SPLINE
SPL {X  -103.775, Y  +255.731, Z    +0.000, E1   +56.205, E3 +52331.695}
SPL {X  -141.196, Y  +302.265, Z    +0.000, E1   +49.914, E3 +52369.180}
SPL {X  -155.405, Y  +339.473, Z    +0.000, E1   +34.418, E3 +52378.880}
SPL {X  -159.172, Y  +361.346, Z    +0.000, E1   +18.323, E3 +52381.305}
SPL {X  -159.962, Y  +374.520, Z    +0.000, E1    +5.534, E3 +52381.918}
SPL {X  -159.990, Y  +379.490, Z    +0.000, E1    +0.023, E3 +52381.975}
SPL {X  -159.990, Y  +381.667, Z    +0.000, E1    -4.707, E3 +52381.997}
SPL {X  -159.990, Y  +385.814, Z    +0.000, E1   -15.621, E3 +52382.101}
SPL {X  -159.990, Y  +390.948, Z    +0.000, E1   -28.850, E3 +52382.377}
SPL {X  -159.990, Y  +399.006, Z    +0.000, E1   -45.565, E3 +52383.089}
SPL {X  -159.990, Y  +410.008, Z    +0.000, E1   -58.546, E3 +52384.699}
SPL {X  -159.990, Y  +426.664, Z    +0.000, E1   -66.963, E3 +52388.320}
SPL {X  -159.990, Y  +494.829, Z    +0.000, E1   -73.764, E3 +52410.084}
SPL {X  -158.798, Y  +695.991, Z    +0.000, E1   -74.986, E3 +52500.017}
SPL {X  -156.512, Y  +709.677, Z    +0.000, E1   -74.772, E3 +52510.161}
SPL {X  -153.684, Y  +720.975, Z    +0.000, E1   -74.508, E3 +52519.448}
SPL {X  -149.353, Y  +733.863, Z    +0.000, E1   -74.100, E3 +52531.036}
SPL {X  -145.190, Y  +743.705, Z    +0.000, E1   -73.640, E3 +52540.717}
SPL {X  -141.940, Y  +750.322, Z    +0.000, E1   -73.290, E3 +52547.484}
SPL {X  -138.555, Y  +756.496, Z    +0.000, E1   -72.905, E3 +52554.049}
SPL {X  -135.025, Y  +762.319, Z    +0.000, E1   -72.483, E3 +52560.428}
SPL {X  -131.747, Y  +767.272, Z    +0.000, E1   -72.071, E3 +52565.953}
SPL {X  -128.648, Y  +771.613, Z    +0.000, E1   -71.666, E3 +52570.845}
SPL {X  -125.012, Y  +776.344, Z    +0.000, E1   -71.184, E3 +52576.157}
SPL {X  -121.578, Y  +780.498, Z    +0.000, E1   -70.681, E3 +52580.800}
SPL {X  -119.460, Y  +782.925, Z    +0.000, E1   -70.353, E3 +52583.464}
SPL {X   -74.295, Y  +818.193, Z    +0.000, E1   -57.793, E3 +52692.125}
ENDSPLINE

SPLINE
SPL {X  -120.240, Y  +782.043, Z    +0.000, E1   -55.019, E3 +52890.621}
SPL {X  -145.777, Y  +742.423, Z    +0.000, E1   -46.722, E3 +52912.501}
SPL {X  -154.920, Y  +716.458, Z    +0.000, E1   -35.175, E3 +52918.556}
SPL {X  -159.063, Y  +693.702, Z    +0.000, E1   -19.028, E3 +52921.337}
SPL {X  -159.958, Y  +679.684, Z    +0.000, E1    -5.688, E3 +52922.049}
SPL {X  -159.990, Y  +674.512, Z    +0.000, E1    -0.026, E3 +52922.114}
SPL {X  -159.990, Y  +672.767, Z    +0.000, E1    +3.705, E3 +52922.127}
SPL {X  -159.990, Y  +669.310, Z    +0.000, E1   +12.444, E3 +52922.201}
SPL {X  -159.990, Y  +665.511, Z    +0.000, E1   +22.359, E3 +52922.360}
SPL {X  -159.990, Y  +658.432, Z    +0.000, E1   +38.720, E3 +52922.884}
SPL {X  -159.990, Y  +646.280, Z    +0.000, E1   +56.156, E3 +52924.413}
SPL {X  -159.990, Y  +625.549, Z    +0.000, E1   +67.208, E3 +52928.935}
SPL {X  -159.990, Y  +550.186, Z    +0.000, E1   +73.637, E3 +52954.340}
SPL {X  -159.493, Y  +364.902, Z    +0.000, E1   +74.541, E3 +53041.334}
SPL {X  -156.915, Y  +346.281, Z    +0.000, E1   +74.304, E3 +53054.930}
ENDSPLINE

SPLINE
SPL {X  -159.697, Y  +367.814, Z    +0.000, E1   +71.217, E3 +53072.248}
ENDSPLINE

SPLINE
SPL {X  -156.028, Y  +342.114, Z    +0.000, E1   +72.020, E3 +53082.402}
SPL {X  -150.925, Y  +324.412, Z    +0.000, E1   +72.419, E3 +53090.195}
SPL {X  -144.972, Y  +309.824, Z    +0.000, E1   +72.799, E3 +53095.797}
SPL {X  -139.605, Y  +299.351, Z    +0.000, E1   +73.035, E3 +53099.928}
SPL {X  -136.475, Y  +294.006, Z    +0.000, E1   +72.670, E3 +53105.713}
SPL {X  -133.214, Y  +288.895, Z    +0.000, E1   +72.272, E3 +53111.361}
SPL {X  -129.829, Y  +284.006, Z    +0.000, E1   +71.844, E3 +53116.836}
SPL {X  -126.314, Y  +279.309, Z    +0.000, E1   +71.374, E3 +53122.128}
SPL {X  -122.705, Y  +274.834, Z    +0.000, E1   +70.869, E3 +53127.139}
SPL {X  -119.804, Y  +271.463, Z    +0.000, E1   +70.429, E3 +53130.858}
SPL {X   -77.409, Y  +237.483, Z    +0.000, E1   +59.013, E3 +53224.534}
ENDSPLINE

SPLINE
SPL {X  -103.775, Y  +255.731, Z    +0.000, E1   +56.205, E3 +53421.247}
SPL {X  -133.021, Y  +288.605, Z    +0.000, E1   +53.007, E3 +53452.703}
SPL {X  -149.384, Y  +320.219, Z    +0.000, E1   +43.953, E3 +53464.427}
SPL {X  -157.534, Y  +349.577, Z    +0.000, E1   +27.748, E3 +53469.779}
SPL {X  -159.460, Y  +364.489, Z    +0.000, E1   +15.407, E3 +53471.074}
SPL {X  -159.962, Y  +374.520, Z    +0.000, E1    +5.534, E3 +53471.470}
SPL {X  -159.990, Y  +379.490, Z    +0.000, E1    +0.023, E3 +53471.527}
SPL {X  -159.990, Y  +381.667, Z    +0.000, E1    -4.707, E3 +53471.549}
SPL {X  -159.990, Y  +387.434, Z    +0.000, E1   -19.600, E3 +53471.732}
SPL {X  -159.990, Y  +392.971, Z    +0.000, E1   -33.903, E3 +53472.065}
SPL {X  -159.990, Y  +399.006, Z    +0.000, E1   -45.565, E3 +53472.641}
SPL {X  -159.990, Y  +410.008, Z    +0.000, E1   -58.546, E3 +53474.251}
SPL {X  -159.990, Y  +426.664, Z    +0.000, E1   -66.963, E3 +53477.872}
SPL {X  -159.990, Y  +494.829, Z    +0.000, E1   -73.764, E3 +53499.637}
SPL {X  -158.798, Y  +695.991, Z    +0.000, E1   -74.986, E3 +53589.569}
SPL {X  -156.512, Y  +709.677, Z    +0.000, E1   -74.772, E3 +53599.713}
SPL {X  -153.684, Y  +720.975, Z    +0.000, E1   -74.508, E3 +53609.000}
SPL {X  -149.353, Y  +733.863, Z    +0.000, E1   -74.100, E3 +53620.588}
SPL {X  -145.190, Y  +743.705, Z    +0.000, E1   -73.640, E3 +53630.269}
SPL {X  -141.940, Y  +750.322, Z    +0.000, E1   -73.290, E3 +53637.036}
SPL {X  -138.555, Y  +756.496, Z    +0.000, E1   -72.905, E3 +53643.601}
SPL {X  -135.025, Y  +762.319, Z    +0.000, E1   -72.483, E3 +53649.980}
SPL {X  -131.747, Y  +767.272, Z    +0.000, E1   -72.071, E3 +53655.505}
SPL {X  -127.432, Y  +773.236, Z    +0.000, E1   -71.530, E3 +53662.191}
SPL {X  -124.036, Y  +777.554, Z    +0.000, E1   -71.026, E3 +53667.089}
SPL {X  -120.782, Y  +781.422, Z    +0.000, E1   -70.584, E3 +53671.347}
SPL {X   -74.295, Y  +818.193, Z    +0.000, E1   -57.793, E3 +53781.678}
ENDSPLINE

SPLINE
SPL {X  -105.102, Y  +797.125, Z    +0.000, E1   -55.734, E3 +53961.044}
SPL {X  -126.361, Y  +774.631, Z    +0.000, E1   -54.192, E3 +53986.712}
SPL {X  -145.777, Y  +742.423, Z    +0.000, E1   -46.722, E3 +54002.053}
SPL {X  -154.920, Y  +716.458, Z    +0.000, E1   -35.175, E3 +54008.108}
SPL {X  -159.063, Y  +693.702, Z    +0.000, E1   -19.028, E3 +54010.889}
SPL {X  -159.958, Y  +679.684, Z    +0.000, E1    -5.688, E3 +54011.601}
SPL {X  -159.990, Y  +674.512, Z    +0.000, E1    -0.026, E3 +54011.666}
SPL {X  -159.990, Y  +672.767, Z    +0.000, E1    +3.705, E3 +54011.679}
SPL {X  -159.990, Y  +669.310, Z    +0.000, E1   +12.444, E3 +54011.753}
SPL {X  -159.990, Y  +665.511, Z    +0.000, E1   +22.359, E3 +54011.912}
SPL {X  -159.990, Y  +660.776, Z    +0.000, E1   +34.018, E3 +54012.218}
SPL {X  -159.990, Y  +655.863, Z    +0.000, E1   +43.768, E3 +54012.676}
SPL {X  -159.990, Y  +646.280, Z    +0.000, E1   +56.156, E3 +54013.965}
SPL {X  -159.990, Y  +625.549, Z    +0.000, E1   +67.208, E3 +54018.487}
SPL {X  -159.990, Y  +550.186, Z    +0.000, E1   +73.637, E3 +54043.893}
SPL {X  -159.493, Y  +364.902, Z    +0.000, E1   +74.541, E3 +54130.886}
SPL {X  -156.915, Y  +346.281, Z    +0.000, E1   +74.304, E3 +54144.482}
ENDSPLINE

SPLINE
SPL {X  -159.697, Y  +367.814, Z    +0.000, E1   +71.217, E3 +54161.800}
ENDSPLINE

SPLINE
SPL {X  -157.536, Y  +349.586, Z    +0.000, E1   +71.787, E3 +54169.098}
SPL {X  -154.855, Y  +337.291, Z    +0.000, E1   +72.155, E3 +54173.853}
SPL {X  -150.925, Y  +324.412, Z    +0.000, E1   +72.419, E3 +54179.747}
SPL {X  -146.819, Y  +313.931, Z    +0.000, E1   +72.621, E3 +54184.440}
SPL {X  -140.820, Y  +301.561, Z    +0.000, E1   +73.023, E3 +54188.356}
SPL {X  -136.475, Y  +294.006, Z    +0.000, E1   +72.670, E3 +54195.265}
SPL {X  -133.214, Y  +288.895, Z    +0.000, E1   +72.272, E3 +54200.913}
SPL {X  -129.829, Y  +284.006, Z    +0.000, E1   +71.844, E3 +54206.388}
SPL {X  -126.314, Y  +279.309, Z    +0.000, E1   +71.374, E3 +54211.680}
SPL {X  -122.705, Y  +274.834, Z    +0.000, E1   +70.869, E3 +54216.692}
SPL {X  -119.804, Y  +271.463, Z    +0.000, E1   +70.429, E3 +54220.410}
SPL {X   -77.409, Y  +237.483, Z    +0.000, E1   +59.013, E3 +54314.086}
ENDSPLINE

SPLINE
SPL {X  -103.775, Y  +255.731, Z    +0.000, E1   +56.205, E3 +54510.799}
SPL {X  -141.196, Y  +302.265, Z    +0.000, E1   +49.914, E3 +54548.284}
SPL {X  -155.405, Y  +339.473, Z    +0.000, E1   +34.418, E3 +54557.985}
SPL {X  -159.172, Y  +361.346, Z    +0.000, E1   +18.323, E3 +54560.409}
SPL {X  -159.962, Y  +374.520, Z    +0.000, E1    +5.534, E3 +54561.022}
SPL {X  -159.990, Y  +379.490, Z    +0.000, E1    +0.023, E3 +54561.080}
SPL {X  -159.990, Y  +381.667, Z    +0.000, E1    -4.707, E3 +54561.101}
SPL {X  -159.990, Y  +387.434, Z    +0.000, E1   -19.600, E3 +54561.284}
SPL {X  -159.990, Y  +395.000, Z    +0.000, E1   -38.121, E3 +54561.793}
SPL {X  -159.990, Y  +406.380, Z    +0.000, E1   -55.108, E3 +54563.234}
SPL {X  -159.990, Y  +426.664, Z    +0.000, E1   -66.963, E3 +54567.425}
SPL {X  -159.990, Y  +494.829, Z    +0.000, E1   -73.764, E3 +54589.189}
SPL {X  -158.798, Y  +695.991, Z    +0.000, E1   -74.986, E3 +54679.121}
SPL {X  -156.512, Y  +709.677, Z    +0.000, E1   -74.772, E3 +54689.265}
SPL {X  -153.684, Y  +720.975, Z    +0.000, E1   -74.508, E3 +54698.552}
SPL {X  -149.353, Y  +733.863, Z    +0.000, E1   -74.100, E3 +54710.140}
SPL {X  -145.190, Y  +743.705, Z    +0.000, E1   -73.640, E3 +54719.821}
SPL {X  -141.940, Y  +750.322, Z    +0.000, E1   -73.290, E3 +54726.588}
SPL {X  -138.555, Y  +756.496, Z    +0.000, E1   -72.905, E3 +54733.153}
SPL {X  -135.025, Y  +762.319, Z    +0.000, E1   -72.483, E3 +54739.533}
SPL {X  -131.747, Y  +767.272, Z    +0.000, E1   -72.071, E3 +54745.058}
SPL {X  -127.432, Y  +773.236, Z    +0.000, E1   -71.530, E3 +54751.743}
SPL {X  -124.036, Y  +777.554, Z    +0.000, E1   -71.026, E3 +54756.641}
SPL {X  -120.782, Y  +781.422, Z    +0.000, E1   -70.584, E3 +54760.899}
SPL {X   -74.295, Y  +818.193, Z    +0.000, E1   -57.793, E3 +54871.230}
ENDSPLINE

SPLINE
SPL {X  -105.102, Y  +797.125, Z    +0.000, E1   -55.734, E3 +55050.597}
SPL {X  -126.361, Y  +774.631, Z    +0.000, E1   -54.192, E3 +55076.264}
SPL {X  -145.777, Y  +742.423, Z    +0.000, E1   -46.722, E3 +55091.605}
SPL {X  -154.920, Y  +716.458, Z    +0.000, E1   -35.175, E3 +55097.660}
SPL {X  -158.252, Y  +700.019, Z    +0.000, E1   -24.087, E3 +55099.912}
SPL {X  -159.434, Y  +689.826, Z    +0.000, E1   -15.506, E3 +55100.730}
SPL {X  -159.958, Y  +679.684, Z    +0.000, E1    -5.688, E3 +55101.153}
SPL {X  -159.990, Y  +674.512, Z    +0.000, E1    -0.026, E3 +55101.218}
SPL {X  -159.990, Y  +672.767, Z    +0.000, E1    +3.705, E3 +55101.231}
SPL {X  -159.990, Y  +669.310, Z    +0.000, E1   +12.444, E3 +55101.305}
SPL {X  -159.990, Y  +665.511, Z    +0.000, E1   +22.359, E3 +55101.464}
SPL {X  -159.990, Y  +660.776, Z    +0.000, E1   +34.018, E3 +55101.771}
SPL {X  -159.990, Y  +655.863, Z    +0.000, E1   +43.768, E3 +55102.228}
SPL {X  -159.990, Y  +646.280, Z    +0.000, E1   +56.156, E3 +55103.517}
SPL {X  -159.990, Y  +625.549, Z    +0.000, E1   +67.208, E3 +55108.039}
SPL {X  -159.990, Y  +550.186, Z    +0.000, E1   +73.637, E3 +55133.445}
SPL {X  -159.878, Y  +371.520, Z    +0.000, E1   +74.559, E3 +55216.207}
SPL {X  -159.109, Y  +360.737, Z    +0.000, E1   +74.490, E3 +55223.331}
SPL {X  -156.915, Y  +346.281, Z    +0.000, E1   +74.304, E3 +55234.034}
ENDSPLINE

SPLINE
SPL {X  -159.697, Y  +367.814, Z    +0.000, E1   +71.217, E3 +55251.353}
ENDSPLINE

SPLINE
SPL {X  -156.028, Y  +342.114, Z    +0.000, E1   +72.020, E3 +55261.506}
SPL {X  -150.925, Y  +324.412, Z    +0.000, E1   +72.419, E3 +55269.299}
SPL {X  -146.819, Y  +313.931, Z    +0.000, E1   +72.621, E3 +55273.992}
SPL {X  -140.820, Y  +301.561, Z    +0.000, E1   +73.023, E3 +55277.909}
SPL {X  -136.475, Y  +294.006, Z    +0.000, E1   +72.670, E3 +55284.818}
SPL {X  -133.214, Y  +288.895, Z    +0.000, E1   +72.272, E3 +55290.465}
SPL {X  -129.829, Y  +284.006, Z    +0.000, E1   +71.844, E3 +55295.940}
SPL {X  -125.428, Y  +278.179, Z    +0.000, E1   +71.273, E3 +55302.478}
SPL {X  -120.729, Y  +272.518, Z    +0.000, E1   +70.593, E3 +55308.787}
SPL {X   -77.409, Y  +237.483, Z    +0.000, E1   +59.013, E3 +55403.638}
ENDSPLINE

SPLINE
SPL {X  -103.775, Y  +255.731, Z    +0.000, E1   +56.205, E3 +55600.351}
SPL {X  -141.196, Y  +302.265, Z    +0.000, E1   +49.914, E3 +55637.836}
SPL {X  -155.405, Y  +339.473, Z    +0.000, E1   +34.418, E3 +55647.537}
SPL {X  -159.172, Y  +361.346, Z    +0.000, E1   +18.323, E3 +55649.961}
SPL {X  -159.962, Y  +374.520, Z    +0.000, E1    +5.534, E3 +55650.574}
SPL {X  -159.990, Y  +379.490, Z    +0.000, E1    +0.023, E3 +55650.632}
SPL {X  -159.990, Y  +381.667, Z    +0.000, E1    -4.707, E3 +55650.654}
SPL {X  -159.990, Y  +385.814, Z    +0.000, E1   -15.621, E3 +55650.758}
SPL {X  -159.990, Y  +390.948, Z    +0.000, E1   -28.850, E3 +55651.034}
SPL {X  -159.990, Y  +399.006, Z    +0.000, E1   -45.565, E3 +55651.745}
SPL {X  -159.990, Y  +410.008, Z    +0.000, E1   -58.546, E3 +55653.356}
SPL {X  -159.990, Y  +430.714, Z    +0.000, E1   -67.965, E3 +55658.161}
SPL {X  -159.990, Y  +500.758, Z    +0.000, E1   -73.927, E3 +55680.837}
SPL {X  -158.798, Y  +695.991, Z    +0.000, E1   -74.986, E3 +55768.674}
SPL {X  -156.512, Y  +709.677, Z    +0.000, E1   -74.772, E3 +55778.817}
SPL {X  -153.684, Y  +720.975, Z    +0.000, E1   -74.508, E3 +55788.105}
SPL {X  -150.879, Y  +729.719, Z    +0.000, E1   -74.224, E3 +55795.898}
SPL {X  -148.237, Y  +736.689, Z    +0.000, E1   -73.960, E3 +55802.452}
SPL {X  -145.190, Y  +743.705, Z    +0.000, E1   -73.640, E3 +55809.373}
SPL {X  -141.940, Y  +750.322, Z    +0.000, E1   -73.290, E3 +55816.140}
SPL {X  -138.555, Y  +756.496, Z    +0.000, E1   -72.905, E3 +55822.705}
SPL {X  -135.025, Y  +762.319, Z    +0.000, E1   -72.483, E3 +55829.085}
SPL {X  -131.747, Y  +767.272, Z    +0.000, E1   -72.071, E3 +55834.610}
SPL {X  -127.432, Y  +773.236, Z    +0.000, E1   -71.530, E3 +55841.295}
SPL {X  -124.036, Y  +777.554, Z    +0.000, E1   -71.026, E3 +55846.194}
SPL {X  -120.782, Y  +781.422, Z    +0.000, E1   -70.584, E3 +55850.452}
SPL {X   -74.295, Y  +818.193, Z    +0.000, E1   -57.793, E3 +55960.782}
ENDSPLINE

SPLINE
SPL {X  -105.102, Y  +797.125, Z    +0.000, E1   -55.734, E3 +56140.149}
SPL {X  -126.361, Y  +774.631, Z    +0.000, E1   -54.192, E3 +56165.816}
SPL {X  -145.777, Y  +742.423, Z    +0.000, E1   -46.722, E3 +56181.157}
SPL {X  -154.920, Y  +716.458, Z    +0.000, E1   -35.175, E3 +56187.212}
SPL {X  -158.252, Y  +700.019, Z    +0.000, E1   -24.087, E3 +56189.464}
SPL {X  -159.676, Y  +686.525, Z    +0.000, E1   -12.514, E3 +56190.454}
SPL {X  -159.990, Y  +674.678, Z    +0.000, E1    -0.382, E3 +56190.769}
SPL {X  -159.990, Y  +672.767, Z    +0.000, E1    +3.705, E3 +56190.784}
SPL {X  -159.990, Y  +669.310, Z    +0.000, E1   +12.444, E3 +56190.858}
SPL {X  -159.990, Y  +665.511, Z    +0.000, E1   +22.359, E3 +56191.016}
SPL {X  -159.990, Y  +658.432, Z    +0.000, E1   +38.720, E3 +56191.541}
SPL {X  -159.990, Y  +646.280, Z    +0.000, E1   +56.156, E3 +56193.070}
SPL {X  -159.990, Y  +625.549, Z    +0.000, E1   +67.208, E3 +56197.591}
SPL {X  -159.990, Y  +550.186, Z    +0.000, E1   +73.637, E3 +56222.997}
SPL {X  -159.493, Y  +364.902, Z    +0.000, E1   +74.541, E3 +56309.990}
SPL {X  -156.915, Y  +346.281, Z    +0.000, E1   +74.304, E3 +56323.586}
ENDSPLINE

SPLINE
SPL {X  -159.697, Y  +367.814, Z    +0.000, E1   +71.217, E3 +56340.905}
ENDSPLINE

SPLINE
SPL {X  -156.028, Y  +342.114, Z    +0.000, E1   +72.020, E3 +56351.058}
SPL {X  -150.925, Y  +324.412, Z    +0.000, E1   +72.419, E3 +56358.851}
SPL {X  -144.972, Y  +309.824, Z    +0.000, E1   +72.799, E3 +56364.453}
SPL {X  -139.605, Y  +299.351, Z    +0.000, E1   +73.035, E3 +56368.585}
SPL {X  -136.475, Y  +294.006, Z    +0.000, E1   +72.670, E3 +56374.370}
SPL {X  -133.214, Y  +288.895, Z    +0.000, E1   +72.272, E3 +56380.018}
SPL {X  -129.829, Y  +284.006, Z    +0.000, E1   +71.844, E3 +56385.492}
SPL {X  -126.314, Y  +279.309, Z    +0.000, E1   +71.374, E3 +56390.785}
SPL {X  -122.705, Y  +274.834, Z    +0.000, E1   +70.869, E3 +56395.796}
SPL {X  -119.804, Y  +271.463, Z    +0.000, E1   +70.429, E3 +56399.515}
SPL {X   -77.409, Y  +237.483, Z    +0.000, E1   +59.013, E3 +56493.190}
ENDSPLINE

SPLINE
SPL {X  -103.775, Y  +255.731, Z    +0.000, E1   +56.205, E3 +56689.904}
SPL {X  -133.021, Y  +288.605, Z    +0.000, E1   +53.007, E3 +56721.360}
SPL {X  -149.384, Y  +320.219, Z    +0.000, E1   +43.953, E3 +56733.083}
SPL {X  -157.534, Y  +349.577, Z    +0.000, E1   +27.748, E3 +56738.435}
SPL {X  -159.460, Y  +364.489, Z    +0.000, E1   +15.407, E3 +56739.731}
SPL {X  -159.962, Y  +374.520, Z    +0.000, E1    +5.534, E3 +56740.127}
SPL {X  -159.990, Y  +379.490, Z    +0.000, E1    +0.023, E3 +56740.184}
SPL {X  -159.990, Y  +381.667, Z    +0.000, E1    -4.707, E3 +56740.206}
SPL {X  -159.990, Y  +387.434, Z    +0.000, E1   -19.600, E3 +56740.388}
SPL {X  -159.990, Y  +392.971, Z    +0.000, E1   -33.903, E3 +56740.721}
SPL {X  -159.990, Y  +399.006, Z    +0.000, E1   -45.565, E3 +56741.298}
SPL {X  -159.990, Y  +410.008, Z    +0.000, E1   -58.546, E3 +56742.908}
SPL {X  -159.990, Y  +426.664, Z    +0.000, E1   -66.963, E3 +56746.529}
SPL {X  -159.990, Y  +494.829, Z    +0.000, E1   -73.764, E3 +56768.293}
SPL {X  -158.798, Y  +695.991, Z    +0.000, E1   -74.986, E3 +56858.226}
SPL {X  -156.512, Y  +709.677, Z    +0.000, E1   -74.772, E3 +56868.370}
SPL {X  -153.684, Y  +720.975, Z    +0.000, E1   -74.508, E3 +56877.657}
SPL {X  -149.353, Y  +733.863, Z    +0.000, E1   -74.100, E3 +56889.245}
SPL {X  -145.190, Y  +743.705, Z    +0.000, E1   -73.640, E3 +56898.926}
SPL {X  -141.940, Y  +750.322, Z    +0.000, E1   -73.290, E3 +56905.693}
SPL {X  -138.555, Y  +756.496, Z    +0.000, E1   -72.905, E3 +56912.258}
SPL {X  -135.025, Y  +762.319, Z    +0.000, E1   -72.483, E3 +56918.637}
SPL {X  -131.747, Y  +767.272, Z    +0.000, E1   -72.071, E3 +56924.162}
SPL {X  -128.648, Y  +771.613, Z    +0.000, E1   -71.666, E3 +56929.054}
SPL {X  -125.012, Y  +776.344, Z    +0.000, E1   -71.184, E3 +56934.366}
SPL {X  -121.578, Y  +780.498, Z    +0.000, E1   -70.681, E3 +56939.009}
SPL {X  -119.460, Y  +782.925, Z    +0.000, E1   -70.353, E3 +56941.673}
SPL {X   -74.295, Y  +818.193, Z    +0.000, E1   -57.793, E3 +57050.334}
ENDSPLINE

SPLINE
SPL {X  -120.240, Y  +782.043, Z    +0.000, E1   -55.019, E3 +57248.830}
SPL {X  -145.777, Y  +742.423, Z    +0.000, E1   -46.722, E3 +57270.710}
SPL {X  -154.920, Y  +716.458, Z    +0.000, E1   -35.175, E3 +57276.765}
SPL {X  -159.063, Y  +693.702, Z    +0.000, E1   -19.028, E3 +57279.546}
SPL {X  -159.958, Y  +679.684, Z    +0.000, E1    -5.688, E3 +57280.258}
SPL {X  -159.990, Y  +674.512, Z    +0.000, E1    -0.026, E3 +57280.323}
SPL {X  -159.990, Y  +672.767, Z    +0.000, E1    +3.705, E3 +57280.336}
SPL {X  -159.990, Y  +669.310, Z    +0.000, E1   +12.444, E3 +57280.410}
SPL {X  -159.990, Y  +665.511, Z    +0.000, E1   +22.359, E3 +57280.569}
SPL {X  -159.990, Y  +658.432, Z    +0.000, E1   +38.720, E3 +57281.093}
SPL {X  -159.990, Y  +646.280, Z    +0.000, E1   +56.156, E3 +57282.622}
SPL {X  -159.990, Y  +625.549, Z    +0.000, E1   +67.208, E3 +57287.144}
SPL {X  -159.990, Y  +550.186, Z    +0.000, E1   +73.637, E3 +57312.549}
SPL {X  -159.878, Y  +371.520, Z    +0.000, E1   +74.559, E3 +57395.311}
SPL {X  -159.109, Y  +360.737, Z    +0.000, E1   +74.490, E3 +57402.436}
SPL {X  -156.915, Y  +346.281, Z    +0.000, E1   +74.304, E3 +57413.139}
ENDSPLINE

SPLINE
SPL {X  -159.697, Y  +367.814, Z    +0.000, E1   +71.217, E3 +57430.457}
ENDSPLINE

SPLINE
SPL {X  -157.536, Y  +349.586, Z    +0.000, E1   +71.787, E3 +57437.755}
SPL {X  -154.855, Y  +337.291, Z    +0.000, E1   +72.155, E3 +57442.509}
SPL {X  -150.925, Y  +324.412, Z    +0.000, E1   +72.419, E3 +57448.403}
SPL {X  -146.819, Y  +313.931, Z    +0.000, E1   +72.621, E3 +57453.097}
SPL {X  -140.820, Y  +301.561, Z    +0.000, E1   +73.023, E3 +57457.013}
SPL {X  -136.475, Y  +294.006, Z    +0.000, E1   +72.670, E3 +57463.922}
SPL {X  -133.214, Y  +288.895, Z    +0.000, E1   +72.272, E3 +57469.570}
SPL {X  -129.829, Y  +284.006, Z    +0.000, E1   +71.844, E3 +57475.045}
SPL {X  -126.314, Y  +279.309, Z    +0.000, E1   +71.374, E3 +57480.337}
SPL {X  -122.705, Y  +274.834, Z    +0.000, E1   +70.869, E3 +57485.348}
SPL {X  -119.804, Y  +271.463, Z    +0.000, E1   +70.429, E3 +57489.067}
SPL {X   -77.409, Y  +237.483, Z    +0.000, E1   +59.013, E3 +57582.743}
ENDSPLINE

SPLINE
SPL {X  -103.775, Y  +255.731, Z    +0.000, E1   +56.205, E3 +57779.456}
SPL {X  -141.196, Y  +302.265, Z    +0.000, E1   +49.914, E3 +57816.941}
SPL {X  -153.296, Y  +331.706, Z    +0.000, E1   +38.681, E3 +57825.360}
SPL {X  -157.534, Y  +349.577, Z    +0.000, E1   +27.748, E3 +57827.988}
SPL {X  -159.460, Y  +364.489, Z    +0.000, E1   +15.407, E3 +57829.283}
SPL {X  -159.962, Y  +374.520, Z    +0.000, E1    +5.534, E3 +57829.679}
SPL {X  -159.990, Y  +379.490, Z    +0.000, E1    +0.023, E3 +57829.736}
SPL {X  -159.990, Y  +381.667, Z    +0.000, E1    -4.707, E3 +57829.758}
SPL {X  -159.990, Y  +385.814, Z    +0.000, E1   -15.621, E3 +57829.862}
SPL {X  -159.990, Y  +390.948, Z    +0.000, E1   -28.850, E3 +57830.138}
SPL {X  -159.990, Y  +399.006, Z    +0.000, E1   -45.565, E3 +57830.850}
SPL {X  -159.990, Y  +410.008, Z    +0.000, E1   -58.546, E3 +57832.460}
SPL {X  -159.990, Y  +430.714, Z    +0.000, E1   -67.965, E3 +57837.265}
SPL {X  -159.990, Y  +500.758, Z    +0.000, E1   -73.927, E3 +57859.941}
SPL {X  -158.798, Y  +695.991, Z    +0.000, E1   -74.986, E3 +57947.778}
SPL {X  -156.512, Y  +709.677, Z    +0.000, E1   -74.772, E3 +57957.922}
SPL {X  -153.684, Y  +720.975, Z    +0.000, E1   -74.508, E3 +57967.209}
SPL {X  -150.879, Y  +729.719, Z    +0.000, E1   -74.224, E3 +57975.003}
SPL {X  -148.237, Y  +736.689, Z    +0.000, E1   -73.960, E3 +57981.557}
SPL {X  -145.190, Y  +743.705, Z    +0.000, E1   -73.640, E3 +57988.478}
SPL {X  -141.940, Y  +750.322, Z    +0.000, E1   -73.290, E3 +57995.245}
SPL {X  -138.555, Y  +756.496, Z    +0.000, E1   -72.905, E3 +58001.810}
SPL {X  -135.025, Y  +762.319, Z    +0.000, E1   -72.483, E3 +58008.189}
SPL {X  -131.747, Y  +767.272, Z    +0.000, E1   -72.071, E3 +58013.714}
SPL {X  -127.432, Y  +773.236, Z    +0.000, E1   -71.530, E3 +58020.400}
SPL {X  -124.036, Y  +777.554, Z    +0.000, E1   -71.026, E3 +58025.298}
SPL {X  -120.782, Y  +781.422, Z    +0.000, E1   -70.584, E3 +58029.556}
SPL {X   -74.295, Y  +818.193, Z    +0.000, E1   -57.793, E3 +58139.887}
ENDSPLINE

SPLINE
SPL {X  -120.240, Y  +782.043, Z    +0.000, E1   -55.019, E3 +58338.383}
SPL {X  -145.777, Y  +742.423, Z    +0.000, E1   -46.722, E3 +58360.262}
SPL {X  -154.920, Y  +716.458, Z    +0.000, E1   -35.175, E3 +58366.317}
SPL {X  -158.252, Y  +700.019, Z    +0.000, E1   -24.087, E3 +58368.569}
SPL {X  -159.676, Y  +686.525, Z    +0.000, E1   -12.514, E3 +58369.559}
SPL {X  -159.990, Y  +674.678, Z    +0.000, E1    -0.382, E3 +58369.874}
SPL {X  -159.990, Y  +672.767, Z    +0.000, E1    +3.705, E3 +58369.888}
SPL {X  -159.990, Y  +669.310, Z    +0.000, E1   +12.444, E3 +58369.962}
SPL {X  -159.990, Y  +665.511, Z    +0.000, E1   +22.359, E3 +58370.121}
SPL {X  -159.990, Y  +660.776, Z    +0.000, E1   +34.018, E3 +58370.427}
SPL {X  -159.990, Y  +655.863, Z    +0.000, E1   +43.768, E3 +58370.885}
SPL {X  -159.990, Y  +646.280, Z    +0.000, E1   +56.156, E3 +58372.174}
SPL {X  -159.990, Y  +625.549, Z    +0.000, E1   +67.208, E3 +58376.696}
SPL {X  -159.990, Y  +550.186, Z    +0.000, E1   +73.637, E3 +58402.102}
SPL {X  -159.878, Y  +371.520, Z    +0.000, E1   +74.559, E3 +58484.864}
SPL {X  -159.109, Y  +360.737, Z    +0.000, E1   +74.490, E3 +58491.988}
SPL {X  -156.915, Y  +346.281, Z    +0.000, E1   +74.304, E3 +58502.691}
ENDSPLINE

SPLINE
SPL {X  -159.697, Y  +367.814, Z    +0.000, E1   +71.217, E3 +58520.009}
ENDSPLINE

SPLINE
SPL {X  -157.536, Y  +349.586, Z    +0.000, E1   +71.787, E3 +58527.307}
SPL {X  -154.855, Y  +337.291, Z    +0.000, E1   +72.155, E3 +58532.062}
SPL {X  -150.925, Y  +324.412, Z    +0.000, E1   +72.419, E3 +58537.956}
SPL {X  -144.972, Y  +309.824, Z    +0.000, E1   +72.799, E3 +58543.558}
SPL {X  -139.605, Y  +299.351, Z    +0.000, E1   +73.035, E3 +58547.689}
SPL {X  -136.475, Y  +294.006, Z    +0.000, E1   +72.670, E3 +58553.474}
SPL {X  -133.214, Y  +288.895, Z    +0.000, E1   +72.272, E3 +58559.122}
SPL {X  -129.829, Y  +284.006, Z    +0.000, E1   +71.844, E3 +58564.597}
SPL {X  -126.314, Y  +279.309, Z    +0.000, E1   +71.374, E3 +58569.889}
SPL {X  -122.705, Y  +274.834, Z    +0.000, E1   +70.869, E3 +58574.901}
SPL {X  -119.804, Y  +271.463, Z    +0.000, E1   +70.429, E3 +58578.619}
SPL {X   -77.409, Y  +237.483, Z    +0.000, E1   +59.013, E3 +58672.295}
ENDSPLINE

SPLINE
SPL {X  -103.775, Y  +255.731, Z    +0.000, E1   +56.205, E3 +58869.008}
SPL {X  -141.196, Y  +302.265, Z    +0.000, E1   +49.914, E3 +58906.493}
SPL {X  -155.405, Y  +339.473, Z    +0.000, E1   +34.418, E3 +58916.194}
SPL {X  -158.399, Y  +354.990, Z    +0.000, E1   +23.559, E3 +58918.125}
SPL {X  -159.460, Y  +364.489, Z    +0.000, E1   +15.407, E3 +58918.835}
SPL {X  -159.962, Y  +374.520, Z    +0.000, E1    +5.534, E3 +58919.231}
SPL {X  -159.990, Y  +379.490, Z    +0.000, E1    +0.023, E3 +58919.288}
SPL {X  -159.990, Y  +381.667, Z    +0.000, E1    -4.707, E3 +58919.310}
SPL {X  -159.990, Y  +385.814, Z    +0.000, E1   -15.621, E3 +58919.414}
SPL {X  -159.990, Y  +390.948, Z    +0.000, E1   -28.850, E3 +58919.691}
SPL {X  -159.990, Y  +399.006, Z    +0.000, E1   -45.565, E3 +58920.402}
SPL {X  -159.990, Y  +410.008, Z    +0.000, E1   -58.546, E3 +58922.013}
SPL {X  -159.990, Y  +426.664, Z    +0.000, E1   -66.963, E3 +58925.634}
SPL {X  -159.990, Y  +494.829, Z    +0.000, E1   -73.764, E3 +58947.398}
SPL {X  -158.798, Y  +695.991, Z    +0.000, E1   -74.986, E3 +59037.330}
SPL {X  -156.512, Y  +709.677, Z    +0.000, E1   -74.772, E3 +59047.474}
SPL {X  -153.684, Y  +720.975, Z    +0.000, E1   -74.508, E3 +59056.761}
SPL {X  -149.353, Y  +733.863, Z    +0.000, E1   -74.100, E3 +59068.349}
SPL {X  -145.190, Y  +743.705, Z    +0.000, E1   -73.640, E3 +59078.030}
SPL {X  -141.940, Y  +750.322, Z    +0.000, E1   -73.290, E3 +59084.797}
SPL {X  -138.555, Y  +756.496, Z    +0.000, E1   -72.905, E3 +59091.362}
SPL {X  -135.025, Y  +762.319, Z    +0.000, E1   -72.483, E3 +59097.742}
SPL {X  -131.747, Y  +767.272, Z    +0.000, E1   -72.071, E3 +59103.267}
SPL {X  -128.648, Y  +771.613, Z    +0.000, E1   -71.666, E3 +59108.159}
SPL {X  -125.012, Y  +776.344, Z    +0.000, E1   -71.184, E3 +59113.470}
SPL {X  -120.782, Y  +781.422, Z    +0.000, E1   -70.584, E3 +59119.108}
SPL {X   -74.295, Y  +818.193, Z    +0.000, E1   -57.793, E3 +59229.439}
ENDSPLINE

SPLINE
SPL {X  -120.240, Y  +782.043, Z    +0.000, E1   -55.019, E3 +59427.935}
SPL {X  -145.777, Y  +742.423, Z    +0.000, E1   -46.722, E3 +59449.814}
SPL {X  -154.920, Y  +716.458, Z    +0.000, E1   -35.175, E3 +59455.869}
SPL {X  -159.063, Y  +693.702, Z    +0.000, E1   -19.028, E3 +59458.651}
SPL {X  -159.958, Y  +679.684, Z    +0.000, E1    -5.688, E3 +59459.362}
SPL {X  -159.990, Y  +674.512, Z    +0.000, E1    -0.026, E3 +59459.427}
SPL {X  -159.990, Y  +672.767, Z    +0.000, E1    +3.705, E3 +59459.440}
SPL {X  -159.990, Y  +669.310, Z    +0.000, E1   +12.444, E3 +59459.514}
SPL {X  -159.990, Y  +665.511, Z    +0.000, E1   +22.359, E3 +59459.673}
SPL {X  -159.990, Y  +658.432, Z    +0.000, E1   +38.720, E3 +59460.198}
SPL {X  -159.990, Y  +646.280, Z    +0.000, E1   +56.156, E3 +59461.726}
SPL {X  -159.990, Y  +625.549, Z    +0.000, E1   +67.208, E3 +59466.248}
SPL {X  -159.990, Y  +550.186, Z    +0.000, E1   +73.637, E3 +59491.654}
SPL {X  -159.493, Y  +364.902, Z    +0.000, E1   +74.541, E3 +59578.647}
SPL {X  -156.915, Y  +346.281, Z    +0.000, E1   +74.304, E3 +59592.243}
ENDSPLINE

SPLINE
SPL {X  -159.697, Y  +367.814, Z    +0.000, E1   +71.217, E3 +59609.562}
ENDSPLINE

SPLINE
SPL {X  -157.536, Y  +349.586, Z    +0.000, E1   +71.787, E3 +59616.860}
SPL {X  -154.855, Y  +337.291, Z    +0.000, E1   +72.155, E3 +59621.614}
SPL {X  -150.925, Y  +324.412, Z    +0.000, E1   +72.419, E3 +59627.508}
SPL {X  -144.972, Y  +309.824, Z    +0.000, E1   +72.799, E3 +59633.110}
SPL {X  -139.605, Y  +299.351, Z    +0.000, E1   +73.035, E3 +59637.242}
SPL {X  -136.475, Y  +294.006, Z    +0.000, E1   +72.670, E3 +59643.027}
SPL {X  -133.214, Y  +288.895, Z    +0.000, E1   +72.272, E3 +59648.674}
SPL {X  -129.829, Y  +284.006, Z    +0.000, E1   +71.844, E3 +59654.149}
SPL {X  -125.428, Y  +278.179, Z    +0.000, E1   +71.273, E3 +59660.687}
SPL {X  -120.729, Y  +272.518, Z    +0.000, E1   +70.593, E3 +59666.996}
SPL {X   -77.409, Y  +237.483, Z    +0.000, E1   +59.013, E3 +59761.847}
ENDSPLINE

SPLINE
SPL {X  -103.775, Y  +255.731, Z    +0.000, E1   +56.205, E3 +59958.560}
SPL {X  -141.196, Y  +302.265, Z    +0.000, E1   +49.914, E3 +59996.045}
SPL {X  -155.405, Y  +339.473, Z    +0.000, E1   +34.418, E3 +60005.746}
SPL {X  -159.172, Y  +361.346, Z    +0.000, E1   +18.323, E3 +60008.170}
SPL {X  -159.962, Y  +374.520, Z    +0.000, E1    +5.534, E3 +60008.783}
SPL {X  -159.990, Y  +379.490, Z    +0.000, E1    +0.023, E3 +60008.841}
SPL {X  -159.990, Y  +381.667, Z    +0.000, E1    -4.707, E3 +60008.863}
SPL {X  -159.990, Y  +385.814, Z    +0.000, E1   -15.621, E3 +60008.966}
SPL {X  -159.990, Y  +390.948, Z    +0.000, E1   -28.850, E3 +60009.243}
SPL {X  -159.990, Y  +399.006, Z    +0.000, E1   -45.565, E3 +60009.954}
SPL {X  -159.990, Y  +410.008, Z    +0.000, E1   -58.546, E3 +60011.565}
SPL {X  -159.990, Y  +426.664, Z    +0.000, E1   -66.963, E3 +60015.186}
SPL {X  -159.990, Y  +494.829, Z    +0.000, E1   -73.764, E3 +60036.950}
SPL {X  -158.798, Y  +695.991, Z    +0.000, E1   -74.986, E3 +60126.883}
SPL {X  -156.512, Y  +709.677, Z    +0.000, E1   -74.772, E3 +60137.026}
SPL {X  -153.684, Y  +720.975, Z    +0.000, E1   -74.508, E3 +60146.314}
SPL {X  -150.879, Y  +729.719, Z    +0.000, E1   -74.224, E3 +60154.107}
SPL {X  -148.237, Y  +736.689, Z    +0.000, E1   -73.960, E3 +60160.661}
SPL {X  -145.190, Y  +743.705, Z    +0.000, E1   -73.640, E3 +60167.582}
SPL {X  -141.940, Y  +750.322, Z    +0.000, E1   -73.290, E3 +60174.349}
SPL {X  -138.555, Y  +756.496, Z    +0.000, E1   -72.905, E3 +60180.914}
SPL {X  -135.025, Y  +762.319, Z    +0.000, E1   -72.483, E3 +60187.294}
SPL {X  -131.747, Y  +767.272, Z    +0.000, E1   -72.071, E3 +60192.819}
SPL {X  -127.432, Y  +773.236, Z    +0.000, E1   -71.530, E3 +60199.504}
SPL {X  -124.036, Y  +777.554, Z    +0.000, E1   -71.026, E3 +60204.403}
SPL {X  -120.782, Y  +781.422, Z    +0.000, E1   -70.584, E3 +60208.661}
SPL {X   -74.295, Y  +818.193, Z    +0.000, E1   -57.793, E3 +60318.991}
ENDSPLINE

SPLINE
SPL {X  -105.102, Y  +797.125, Z    +0.000, E1   -55.734, E3 +60498.358}
SPL {X  -126.361, Y  +774.631, Z    +0.000, E1   -54.192, E3 +60524.025}
SPL {X  -145.777, Y  +742.423, Z    +0.000, E1   -46.722, E3 +60539.366}
SPL {X  -154.920, Y  +716.458, Z    +0.000, E1   -35.175, E3 +60545.421}
SPL {X  -159.063, Y  +693.702, Z    +0.000, E1   -19.028, E3 +60548.203}
SPL {X  -159.958, Y  +679.684, Z    +0.000, E1    -5.688, E3 +60548.915}
SPL {X  -159.990, Y  +674.512, Z    +0.000, E1    -0.026, E3 +60548.979}
SPL {X  -159.990, Y  +672.767, Z    +0.000, E1    +3.705, E3 +60548.993}
SPL {X  -159.990, Y  +669.310, Z    +0.000, E1   +12.444, E3 +60549.067}
SPL {X  -159.990, Y  +665.511, Z    +0.000, E1   +22.359, E3 +60549.225}
SPL {X  -159.990, Y  +660.776, Z    +0.000, E1   +34.018, E3 +60549.532}
SPL {X  -159.990, Y  +655.863, Z    +0.000, E1   +43.768, E3 +60549.989}
SPL {X  -159.990, Y  +646.280, Z    +0.000, E1   +56.156, E3 +60551.279}
SPL {X  -159.990, Y  +625.549, Z    +0.000, E1   +67.208, E3 +60555.800}
SPL {X  -159.990, Y  +550.186, Z    +0.000, E1   +73.637, E3 +60581.206}
SPL {X  -159.493, Y  +364.902, Z    +0.000, E1   +74.541, E3 +60668.199}
SPL {X  -156.915, Y  +346.281, Z    +0.000, E1   +74.304, E3 +60681.795}
ENDSPLINE

SPLINE
SPL {X  -159.697, Y  +367.814, Z    +0.000, E1   +71.217, E3 +60699.114}
ENDSPLINE

SPLINE
SPL {X  -157.536, Y  +349.586, Z    +0.000, E1   +71.787, E3 +60706.412}
SPL {X  -154.855, Y  +337.291, Z    +0.000, E1   +72.155, E3 +60711.166}
SPL {X  -150.925, Y  +324.412, Z    +0.000, E1   +72.419, E3 +60717.060}
SPL {X  -146.819, Y  +313.931, Z    +0.000, E1   +72.621, E3 +60721.754}
SPL {X  -140.820, Y  +301.561, Z    +0.000, E1   +73.023, E3 +60725.670}
SPL {X  -136.475, Y  +294.006, Z    +0.000, E1   +72.670, E3 +60732.579}
SPL {X  -133.214, Y  +288.895, Z    +0.000, E1   +72.272, E3 +60738.227}
SPL {X  -129.829, Y  +284.006, Z    +0.000, E1   +71.844, E3 +60743.701}
SPL {X  -126.314, Y  +279.309, Z    +0.000, E1   +71.374, E3 +60748.994}
SPL {X  -122.705, Y  +274.834, Z    +0.000, E1   +70.869, E3 +60754.005}
SPL {X  -119.804, Y  +271.463, Z    +0.000, E1   +70.429, E3 +60757.724}
SPL {X   -77.409, Y  +237.483, Z    +0.000, E1   +59.013, E3 +60851.399}
ENDSPLINE

SPLINE
SPL {X  -103.775, Y  +255.731, Z    +0.000, E1   +56.205, E3 +61048.113}
SPL {X  -141.196, Y  +302.265, Z    +0.000, E1   +49.914, E3 +61085.598}
SPL {X  -155.405, Y  +339.473, Z    +0.000, E1   +34.418, E3 +61095.298}
SPL {X  -159.172, Y  +361.346, Z    +0.000, E1   +18.323, E3 +61097.723}
SPL {X  -159.962, Y  +374.520, Z    +0.000, E1    +5.534, E3 +61098.336}
SPL {X  -159.990, Y  +379.490, Z    +0.000, E1    +0.023, E3 +61098.393}
SPL {X  -159.990, Y  +381.667, Z    +0.000, E1    -4.707, E3 +61098.415}
SPL {X  -159.990, Y  +387.434, Z    +0.000, E1   -19.600, E3 +61098.597}
SPL {X  -159.990, Y  +395.000, Z    +0.000, E1   -38.121, E3 +61099.106}
SPL {X  -159.990, Y  +406.380, Z    +0.000, E1   -55.108, E3 +61100.548}
SPL {X  -159.990, Y  +426.664, Z    +0.000, E1   -66.963, E3 +61104.738}
SPL {X  -159.990, Y  +494.829, Z    +0.000, E1   -73.764, E3 +61126.502}
SPL {X  -158.798, Y  +695.991, Z    +0.000, E1   -74.986, E3 +61216.435}
SPL {X  -156.512, Y  +709.677, Z    +0.000, E1   -74.772, E3 +61226.578}
SPL {X  -153.684, Y  +720.975, Z    +0.000, E1   -74.508, E3 +61235.866}
SPL {X  -149.353, Y  +733.863, Z    +0.000, E1   -74.100, E3 +61247.454}
SPL {X  -145.190, Y  +743.705, Z    +0.000, E1   -73.640, E3 +61257.135}
SPL {X  -141.940, Y  +750.322, Z    +0.000, E1   -73.290, E3 +61263.901}
SPL {X  -138.555, Y  +756.496, Z    +0.000, E1   -72.905, E3 +61270.466}
SPL {X  -135.025, Y  +762.319, Z    +0.000, E1   -72.483, E3 +61276.846}
SPL {X  -131.747, Y  +767.272, Z    +0.000, E1   -72.071, E3 +61282.371}
SPL {X  -127.432, Y  +773.236, Z    +0.000, E1   -71.530, E3 +61289.056}
SPL {X  -124.036, Y  +777.554, Z    +0.000, E1   -71.026, E3 +61293.955}
SPL {X  -120.782, Y  +781.422, Z    +0.000, E1   -70.584, E3 +61298.213}
SPL {X   -74.295, Y  +818.193, Z    +0.000, E1   -57.793, E3 +61408.543}
ENDSPLINE

SPLINE
SPL {X  -105.102, Y  +797.125, Z    +0.000, E1   -55.734, E3 +61587.910}
SPL {X  -126.361, Y  +774.631, Z    +0.000, E1   -54.192, E3 +61613.578}
SPL {X  -145.777, Y  +742.423, Z    +0.000, E1   -46.722, E3 +61628.919}
SPL {X  -154.920, Y  +716.458, Z    +0.000, E1   -35.175, E3 +61634.974}
SPL {X  -159.063, Y  +693.702, Z    +0.000, E1   -19.028, E3 +61637.755}
SPL {X  -159.958, Y  +679.684, Z    +0.000, E1    -5.688, E3 +61638.467}
SPL {X  -159.990, Y  +674.512, Z    +0.000, E1    -0.026, E3 +61638.532}
SPL {X  -159.990, Y  +672.767, Z    +0.000, E1    +3.705, E3 +61638.545}
SPL {X  -159.990, Y  +669.310, Z    +0.000, E1   +12.444, E3 +61638.619}
SPL {X  -159.990, Y  +665.511, Z    +0.000, E1   +22.359, E3 +61638.778}
SPL {X  -159.990, Y  +660.776, Z    +0.000, E1   +34.018, E3 +61639.084}
SPL {X  -159.990, Y  +655.863, Z    +0.000, E1   +43.768, E3 +61639.542}
SPL {X  -159.990, Y  +646.280, Z    +0.000, E1   +56.156, E3 +61640.831}
SPL {X  -159.990, Y  +625.549, Z    +0.000, E1   +67.208, E3 +61645.353}
SPL {X  -159.990, Y  +550.186, Z    +0.000, E1   +73.637, E3 +61670.758}
SPL {X  -159.493, Y  +364.902, Z    +0.000, E1   +74.541, E3 +61757.752}
SPL {X  -156.915, Y  +346.281, Z    +0.000, E1   +74.304, E3 +61771.348}
ENDSPLINE

SPLINE
SPL {X  -159.697, Y  +367.814, Z    +0.000, E1   +71.217, E3 +61788.666}
ENDSPLINE

SPLINE
SPL {X  -156.028, Y  +342.114, Z    +0.000, E1   +72.020, E3 +61798.820}
SPL {X  -150.925, Y  +324.412, Z    +0.000, E1   +72.419, E3 +61806.612}
SPL {X  -144.972, Y  +309.824, Z    +0.000, E1   +72.799, E3 +61812.214}
SPL {X  -139.605, Y  +299.351, Z    +0.000, E1   +73.035, E3 +61816.346}
SPL {X  -136.475, Y  +294.006, Z    +0.000, E1   +72.670, E3 +61822.131}
SPL {X  -133.214, Y  +288.895, Z    +0.000, E1   +72.272, E3 +61827.779}
SPL {X  -129.829, Y  +284.006, Z    +0.000, E1   +71.844, E3 +61833.254}
SPL {X  -125.428, Y  +278.179, Z    +0.000, E1   +71.273, E3 +61839.791}
SPL {X  -120.729, Y  +272.518, Z    +0.000, E1   +70.593, E3 +61846.101}
SPL {X   -77.409, Y  +237.483, Z    +0.000, E1   +59.013, E3 +61940.951}
ENDSPLINE

SPLINE
SPL {X  -103.775, Y  +255.731, Z    +0.000, E1   +56.205, E3 +62137.665}
SPL {X  -141.196, Y  +302.265, Z    +0.000, E1   +49.914, E3 +62175.150}
SPL {X  -153.296, Y  +331.706, Z    +0.000, E1   +38.681, E3 +62183.569}
SPL {X  -157.534, Y  +349.577, Z    +0.000, E1   +27.748, E3 +62186.197}
SPL {X  -159.460, Y  +364.489, Z    +0.000, E1   +15.407, E3 +62187.492}
SPL {X  -159.962, Y  +374.520, Z    +0.000, E1    +5.534, E3 +62187.888}
SPL {X  -159.990, Y  +379.490, Z    +0.000, E1    +0.023, E3 +62187.945}
SPL {X  -159.990, Y  +381.667, Z    +0.000, E1    -4.707, E3 +62187.967}
SPL {X  -159.990, Y  +387.434, Z    +0.000, E1   -19.600, E3 +62188.150}
SPL {X  -159.990, Y  +392.971, Z    +0.000, E1   -33.903, E3 +62188.482}
SPL {X  -159.990, Y  +399.006, Z    +0.000, E1   -45.565, E3 +62189.059}
SPL {X  -159.990, Y  +410.008, Z    +0.000, E1   -58.546, E3 +62190.669}
SPL {X  -159.990, Y  +426.664, Z    +0.000, E1   -66.963, E3 +62194.290}
SPL {X  -159.990, Y  +494.829, Z    +0.000, E1   -73.764, E3 +62216.054}
SPL {X  -158.798, Y  +695.991, Z    +0.000, E1   -74.986, E3 +62305.987}
SPL {X  -156.512, Y  +709.677, Z    +0.000, E1   -74.772, E3 +62316.131}
SPL {X  -153.684, Y  +720.975, Z    +0.000, E1   -74.508, E3 +62325.418}
SPL {X  -149.353, Y  +733.863, Z    +0.000, E1   -74.100, E3 +62337.006}
SPL {X  -145.190, Y  +743.705, Z    +0.000, E1   -73.640, E3 +62346.687}
SPL {X  -141.940, Y  +750.322, Z    +0.000, E1   -73.290, E3 +62353.454}
SPL {X  -138.555, Y  +756.496, Z    +0.000, E1   -72.905, E3 +62360.019}
SPL {X  -135.025, Y  +762.319, Z    +0.000, E1   -72.483, E3 +62366.398}
SPL {X  -131.747, Y  +767.272, Z    +0.000, E1   -72.071, E3 +62371.923}
SPL {X  -127.432, Y  +773.236, Z    +0.000, E1   -71.530, E3 +62378.609}
SPL {X  -124.036, Y  +777.554, Z    +0.000, E1   -71.026, E3 +62383.507}
SPL {X  -120.782, Y  +781.422, Z    +0.000, E1   -70.584, E3 +62387.765}
SPL {X   -74.295, Y  +818.193, Z    +0.000, E1   -57.793, E3 +62498.096}
ENDSPLINE

SPLINE
SPL {X  -105.102, Y  +797.125, Z    +0.000, E1   -55.734, E3 +62677.462}
SPL {X  -126.361, Y  +774.631, Z    +0.000, E1   -54.192, E3 +62703.130}
SPL {X  -145.777, Y  +742.423, Z    +0.000, E1   -46.722, E3 +62718.471}
SPL {X  -154.920, Y  +716.458, Z    +0.000, E1   -35.175, E3 +62724.526}
SPL {X  -158.252, Y  +700.019, Z    +0.000, E1   -24.087, E3 +62726.778}
SPL {X  -159.676, Y  +686.525, Z    +0.000, E1   -12.514, E3 +62727.768}
SPL {X  -159.990, Y  +674.678, Z    +0.000, E1    -0.382, E3 +62728.083}
SPL {X  -159.990, Y  +672.767, Z    +0.000, E1    +3.705, E3 +62728.097}
SPL {X  -159.990, Y  +669.310, Z    +0.000, E1   +12.444, E3 +62728.171}
SPL {X  -159.990, Y  +665.511, Z    +0.000, E1   +22.359, E3 +62728.330}
SPL {X  -159.990, Y  +658.432, Z    +0.000, E1   +38.720, E3 +62728.855}
SPL {X  -159.990, Y  +646.280, Z    +0.000, E1   +56.156, E3 +62730.383}
SPL {X  -159.990, Y  +625.549, Z    +0.000, E1   +67.208, E3 +62734.905}
SPL {X  -159.990, Y  +550.186, Z    +0.000, E1   +73.637, E3 +62760.311}
SPL {X  -159.878, Y  +371.520, Z    +0.000, E1   +74.559, E3 +62843.073}
SPL {X  -158.372, Y  +354.804, Z    +0.000, E1   +74.445, E3 +62854.377}
SPL {X  -156.009, Y  +342.031, Z    +0.000, E1   +74.195, E3 +62864.387}
ENDSPLINE

SPLINE
SPL {X  -159.697, Y  +367.814, Z    +0.000, E1   +71.217, E3 +62878.218}
ENDSPLINE

SPLINE
SPL {X  -156.028, Y  +342.114, Z    +0.000, E1   +72.020, E3 +62888.372}
SPL {X  -150.925, Y  +324.412, Z    +0.000, E1   +72.419, E3 +62896.165}
SPL {X  -144.972, Y  +309.824, Z    +0.000, E1   +72.799, E3 +62901.767}
SPL {X  -139.605, Y  +299.351, Z    +0.000, E1   +73.035, E3 +62905.898}
SPL {X  -136.475, Y  +294.006, Z    +0.000, E1   +72.670, E3 +62911.683}
SPL {X  -133.214, Y  +288.895, Z    +0.000, E1   +72.272, E3 +62917.331}
SPL {X  -129.829, Y  +284.006, Z    +0.000, E1   +71.844, E3 +62922.806}
SPL {X  -125.428, Y  +278.179, Z    +0.000, E1   +71.273, E3 +62929.343}
SPL {X  -120.729, Y  +272.518, Z    +0.000, E1   +70.593, E3 +62935.653}
SPL {X   -77.409, Y  +237.483, Z    +0.000, E1   +59.013, E3 +63030.504}
ENDSPLINE

SPLINE
SPL {X  -103.775, Y  +255.731, Z    +0.000, E1   +56.205, E3 +63227.217}
SPL {X  -133.021, Y  +288.605, Z    +0.000, E1   +53.007, E3 +63258.673}
SPL {X  -149.384, Y  +320.219, Z    +0.000, E1   +43.953, E3 +63270.397}
SPL {X  -157.534, Y  +349.577, Z    +0.000, E1   +27.748, E3 +63275.749}
SPL {X  -159.460, Y  +364.489, Z    +0.000, E1   +15.407, E3 +63277.044}
SPL {X  -159.962, Y  +374.520, Z    +0.000, E1    +5.534, E3 +63277.440}
SPL {X  -159.990, Y  +379.741, Z    +0.000, E1    -0.257, E3 +63277.499}
SPL {X  -159.990, Y  +384.604, Z    +0.000, E1   -12.124, E3 +63277.588}
SPL {X  -159.990, Y  +389.475, Z    +0.000, E1   -25.351, E3 +63277.801}
SPL {X  -159.990, Y  +395.000, Z    +0.000, E1   -38.121, E3 +63278.211}
SPL {X  -159.990, Y  +406.380, Z    +0.000, E1   -55.108, E3 +63279.652}
SPL {X  -159.990, Y  +426.664, Z    +0.000, E1   -66.963, E3 +63283.843}
SPL {X  -159.990, Y  +494.829, Z    +0.000, E1   -73.764, E3 +63305.607}
SPL {X  -158.798, Y  +695.991, Z    +0.000, E1   -74.986, E3 +63395.539}
SPL {X  -156.512, Y  +709.677, Z    +0.000, E1   -74.772, E3 +63405.683}
SPL {X  -153.684, Y  +720.975, Z    +0.000, E1   -74.508, E3 +63414.970}
SPL {X  -149.353, Y  +733.863, Z    +0.000, E1   -74.100, E3 +63426.558}
SPL {X  -145.190, Y  +743.705, Z    +0.000, E1   -73.640, E3 +63436.239}
SPL {X  -141.940, Y  +750.322, Z    +0.000, E1   -73.290, E3 +63443.006}
SPL {X  -138.555, Y  +756.496, Z    +0.000, E1   -72.905, E3 +63449.571}
SPL {X  -135.025, Y  +762.319, Z    +0.000, E1   -72.483, E3 +63455.951}
SPL {X  -131.747, Y  +767.272, Z    +0.000, E1   -72.071, E3 +63461.476}
SPL {X  -127.432, Y  +773.236, Z    +0.000, E1   -71.530, E3 +63468.161}
SPL {X  -124.036, Y  +777.554, Z    +0.000, E1   -71.026, E3 +63473.059}
SPL {X  -120.782, Y  +781.422, Z    +0.000, E1   -70.584, E3 +63477.317}
SPL {X   -74.295, Y  +818.193, Z    +0.000, E1   -57.793, E3 +63587.648}
ENDSPLINE

SPLINE
SPL {X  -120.240, Y  +782.043, Z    +0.000, E1   -55.019, E3 +63786.144}
SPL {X  -145.777, Y  +742.423, Z    +0.000, E1   -46.722, E3 +63808.023}
SPL {X  -154.920, Y  +716.458, Z    +0.000, E1   -35.175, E3 +63814.078}
SPL {X  -158.252, Y  +700.019, Z    +0.000, E1   -24.087, E3 +63816.330}
SPL {X  -159.676, Y  +686.525, Z    +0.000, E1   -12.514, E3 +63817.320}
SPL {X  -159.990, Y  +674.678, Z    +0.000, E1    -0.382, E3 +63817.635}
SPL {X  -159.990, Y  +672.767, Z    +0.000, E1    +3.705, E3 +63817.649}
SPL {X  -159.990, Y  +669.310, Z    +0.000, E1   +12.444, E3 +63817.723}
SPL {X  -159.990, Y  +665.511, Z    +0.000, E1   +22.359, E3 +63817.882}
SPL {X  -159.990, Y  +660.776, Z    +0.000, E1   +34.018, E3 +63818.189}
SPL {X  -159.990, Y  +655.863, Z    +0.000, E1   +43.768, E3 +63818.646}
SPL {X  -159.990, Y  +646.280, Z    +0.000, E1   +56.156, E3 +63819.935}
SPL {X  -159.990, Y  +625.549, Z    +0.000, E1   +67.208, E3 +63824.457}
SPL {X  -159.990, Y  +550.186, Z    +0.000, E1   +73.637, E3 +63849.863}
SPL {X  -159.878, Y  +371.520, Z    +0.000, E1   +74.559, E3 +63932.625}
SPL {X  -159.109, Y  +360.737, Z    +0.000, E1   +74.490, E3 +63939.749}
SPL {X  -156.915, Y  +346.281, Z    +0.000, E1   +74.304, E3 +63950.452}
ENDSPLINE

SPLINE
SPL {X  -159.697, Y  +367.814, Z    +0.000, E1   +71.217, E3 +63967.771}
ENDSPLINE

SPLINE
SPL {X  -156.028, Y  +342.114, Z    +0.000, E1   +72.020, E3 +63977.924}
SPL {X  -150.925, Y  +324.412, Z    +0.000, E1   +72.419, E3 +63985.717}
SPL {X  -146.819, Y  +313.931, Z    +0.000, E1   +72.621, E3 +63990.410}
SPL {X  -140.820, Y  +301.561, Z    +0.000, E1   +73.023, E3 +63994.327}
SPL {X  -136.475, Y  +294.006, Z    +0.000, E1   +72.670, E3 +64001.236}
SPL {X  -133.214, Y  +288.895, Z    +0.000, E1   +72.272, E3 +64006.883}
SPL {X  -129.829, Y  +284.006, Z    +0.000, E1   +71.844, E3 +64012.358}
SPL {X  -125.428, Y  +278.179, Z    +0.000, E1   +71.273, E3 +64018.896}
SPL {X  -120.729, Y  +272.518, Z    +0.000, E1   +70.593, E3 +64025.205}
SPL {X   -77.409, Y  +237.483, Z    +0.000, E1   +59.013, E3 +64120.056}
ENDSPLINE

SPLINE
SPL {X  -103.775, Y  +255.731, Z    +0.000, E1   +56.205, E3 +64316.769}
SPL {X  -141.196, Y  +302.265, Z    +0.000, E1   +49.914, E3 +64354.254}
SPL {X  -155.405, Y  +339.473, Z    +0.000, E1   +34.418, E3 +64363.955}
SPL {X  -159.172, Y  +361.346, Z    +0.000, E1   +18.323, E3 +64366.379}
SPL {X  -159.962, Y  +374.520, Z    +0.000, E1    +5.534, E3 +64366.992}
SPL {X  -159.990, Y  +379.490, Z    +0.000, E1    +0.023, E3 +64367.050}
SPL {X  -159.990, Y  +381.667, Z    +0.000, E1    -4.707, E3 +64367.072}
SPL {X  -159.990, Y  +385.814, Z    +0.000, E1   -15.621, E3 +64367.175}
SPL {X  -159.990, Y  +390.948, Z    +0.000, E1   -28.850, E3 +64367.452}
SPL {X  -159.990, Y  +399.006, Z    +0.000, E1   -45.565, E3 +64368.163}
SPL {X  -159.990, Y  +410.008, Z    +0.000, E1   -58.546, E3 +64369.774}
SPL {X  -159.990, Y  +426.664, Z    +0.000, E1   -66.963, E3 +64373.395}
SPL {X  -159.990, Y  +494.829, Z    +0.000, E1   -73.764, E3 +64395.159}
SPL {X  -158.798, Y  +695.991, Z    +0.000, E1   -74.986, E3 +64485.092}
SPL {X  -156.512, Y  +709.677, Z    +0.000, E1   -74.772, E3 +64495.235}
SPL {X  -153.684, Y  +720.975, Z    +0.000, E1   -74.508, E3 +64504.523}
SPL {X  -149.353, Y  +733.863, Z    +0.000, E1   -74.100, E3 +64516.110}
SPL {X  -145.190, Y  +743.705, Z    +0.000, E1   -73.640, E3 +64525.791}
SPL {X  -141.940, Y  +750.322, Z    +0.000, E1   -73.290, E3 +64532.558}
SPL {X  -138.555, Y  +756.496, Z    +0.000, E1   -72.905, E3 +64539.123}
SPL {X  -135.025, Y  +762.319, Z    +0.000, E1   -72.483, E3 +64545.503}
SPL {X  -131.747, Y  +767.272, Z    +0.000, E1   -72.071, E3 +64551.028}
SPL {X  -128.648, Y  +771.613, Z    +0.000, E1   -71.666, E3 +64555.920}
SPL {X  -125.012, Y  +776.344, Z    +0.000, E1   -71.184, E3 +64561.232}
SPL {X  -121.578, Y  +780.498, Z    +0.000, E1   -70.681, E3 +64565.875}
SPL {X  -119.460, Y  +782.925, Z    +0.000, E1   -70.353, E3 +64568.539}
SPL {X   -74.295, Y  +818.193, Z    +0.000, E1   -57.793, E3 +64677.200}
ENDSPLINE

SPLINE
SPL {X  -120.240, Y  +782.043, Z    +0.000, E1   -55.019, E3 +64875.696}
SPL {X  -145.777, Y  +742.423, Z    +0.000, E1   -46.722, E3 +64897.575}
SPL {X  -154.920, Y  +716.458, Z    +0.000, E1   -35.175, E3 +64903.630}
SPL {X  -159.063, Y  +693.702, Z    +0.000, E1   -19.028, E3 +64906.412}
SPL {X  -159.958, Y  +679.684, Z    +0.000, E1    -5.688, E3 +64907.124}
SPL {X  -159.990, Y  +674.512, Z    +0.000, E1    -0.026, E3 +64907.188}
SPL {X  -159.990, Y  +672.767, Z    +0.000, E1    +3.705, E3 +64907.202}
SPL {X  -159.990, Y  +669.310, Z    +0.000, E1   +12.444, E3 +64907.276}
SPL {X  -159.990, Y  +665.511, Z    +0.000, E1   +22.359, E3 +64907.434}
SPL {X  -159.990, Y  +658.432, Z    +0.000, E1   +38.720, E3 +64907.959}
SPL {X  -159.990, Y  +646.280, Z    +0.000, E1   +56.156, E3 +64909.488}
SPL {X  -159.990, Y  +625.549, Z    +0.000, E1   +67.208, E3 +64914.009}
SPL {X  -159.990, Y  +550.186, Z    +0.000, E1   +73.637, E3 +64939.415}
SPL {X  -159.493, Y  +364.902, Z    +0.000, E1   +74.541, E3 +65026.408}
SPL {X  -156.915, Y  +346.281, Z    +0.000, E1   +74.304, E3 +65040.004}
ENDSPLINE

SPLINE
SPL {X  -159.697, Y  +367.814, Z    +0.000, E1   +71.217, E3 +65057.323}
ENDSPLINE

SPLINE
SPL {X  -156.028, Y  +342.114, Z    +0.000, E1   +72.020, E3 +65067.476}
SPL {X  -150.925, Y  +324.412, Z    +0.000, E1   +72.419, E3 +65075.269}
SPL {X  -144.972, Y  +309.824, Z    +0.000, E1   +72.799, E3 +65080.871}
SPL {X  -139.605, Y  +299.351, Z    +0.000, E1   +73.035, E3 +65085.003}
SPL {X  -136.475, Y  +294.006, Z    +0.000, E1   +72.670, E3 +65090.788}
SPL {X  -133.214, Y  +288.895, Z    +0.000, E1   +72.272, E3 +65096.436}
SPL {X  -129.829, Y  +284.006, Z    +0.000, E1   +71.844, E3 +65101.910}
SPL {X  -126.314, Y  +279.309, Z    +0.000, E1   +71.374, E3 +65107.203}
SPL {X  -122.705, Y  +274.834, Z    +0.000, E1   +70.869, E3 +65112.214}
SPL {X  -119.804, Y  +271.463, Z    +0.000, E1   +70.429, E3 +65115.933}
SPL {X   -77.409, Y  +237.483, Z    +0.000, E1   +59.013, E3 +65209.608}
ENDSPLINE

SPLINE
SPL {X  -103.775, Y  +255.731, Z    +0.000, E1   +56.205, E3 +65406.321}
SPL {X  -133.021, Y  +288.605, Z    +0.000, E1   +53.007, E3 +65437.778}
SPL {X  -149.384, Y  +320.219, Z    +0.000, E1   +43.953, E3 +65449.501}
SPL {X  -157.534, Y  +349.577, Z    +0.000, E1   +27.748, E3 +65454.853}
SPL {X  -159.460, Y  +364.489, Z    +0.000, E1   +15.407, E3 +65456.149}
SPL {X  -159.962, Y  +374.520, Z    +0.000, E1    +5.534, E3 +65456.545}
SPL {X  -159.990, Y  +379.490, Z    +0.000, E1    +0.023, E3 +65456.602}
SPL {X  -159.990, Y  +381.667, Z    +0.000, E1    -4.707, E3 +65456.624}
SPL {X  -159.990, Y  +387.434, Z    +0.000, E1   -19.600, E3 +65456.806}
SPL {X  -159.990, Y  +392.971, Z    +0.000, E1   -33.903, E3 +65457.139}
SPL {X  -159.990, Y  +399.006, Z    +0.000, E1   -45.565, E3 +65457.716}
SPL {X  -159.990, Y  +410.008, Z    +0.000, E1   -58.546, E3 +65459.326}
SPL {X  -159.990, Y  +426.664, Z    +0.000, E1   -66.963, E3 +65462.947}
SPL {X  -159.990, Y  +494.829, Z    +0.000, E1   -73.764, E3 +65484.711}
SPL {X  -158.798, Y  +695.991, Z    +0.000, E1   -74.986, E3 +65574.644}
SPL {X  -156.512, Y  +709.677, Z    +0.000, E1   -74.772, E3 +65584.787}
SPL {X  -153.684, Y  +720.975, Z    +0.000, E1   -74.508, E3 +65594.075}
SPL {X  -149.353, Y  +733.863, Z    +0.000, E1   -74.100, E3 +65605.663}
SPL {X  -145.190, Y  +743.705, Z    +0.000, E1   -73.640, E3 +65615.344}
SPL {X  -141.940, Y  +750.322, Z    +0.000, E1   -73.290, E3 +65622.110}
SPL {X  -138.555, Y  +756.496, Z    +0.000, E1   -72.905, E3 +65628.675}
SPL {X  -135.025, Y  +762.319, Z    +0.000, E1   -72.483, E3 +65635.055}
SPL {X  -131.747, Y  +767.272, Z    +0.000, E1   -72.071, E3 +65640.580}
SPL {X  -127.432, Y  +773.236, Z    +0.000, E1   -71.530, E3 +65647.265}
SPL {X  -124.036, Y  +777.554, Z    +0.000, E1   -71.026, E3 +65652.164}
SPL {X  -120.782, Y  +781.422, Z    +0.000, E1   -70.584, E3 +65656.422}
SPL {X   -74.295, Y  +818.193, Z    +0.000, E1   -57.793, E3 +65766.752}
ENDSPLINE

SPLINE
SPL {X  -105.102, Y  +797.125, Z    +0.000, E1   -55.734, E3 +65946.119}
SPL {X  -126.361, Y  +774.631, Z    +0.000, E1   -54.192, E3 +65971.787}
SPL {X  -145.777, Y  +742.423, Z    +0.000, E1   -46.722, E3 +65987.128}
SPL {X  -154.920, Y  +716.458, Z    +0.000, E1   -35.175, E3 +65993.183}
SPL {X  -159.063, Y  +693.702, Z    +0.000, E1   -19.028, E3 +65995.964}
SPL {X  -159.958, Y  +679.684, Z    +0.000, E1    -5.688, E3 +65996.676}
SPL {X  -159.990, Y  +674.512, Z    +0.000, E1    -0.026, E3 +65996.740}
SPL {X  -159.990, Y  +672.767, Z    +0.000, E1    +3.705, E3 +65996.754}
SPL {X  -159.990, Y  +669.310, Z    +0.000, E1   +12.444, E3 +65996.828}
SPL {X  -159.990, Y  +665.511, Z    +0.000, E1   +22.359, E3 +65996.986}
SPL {X  -159.990, Y  +660.776, Z    +0.000, E1   +34.018, E3 +65997.293}
SPL {X  -159.990, Y  +655.863, Z    +0.000, E1   +43.768, E3 +65997.750}
SPL {X  -159.990, Y  +646.280, Z    +0.000, E1   +56.156, E3 +65999.040}
SPL {X  -159.990, Y  +625.549, Z    +0.000, E1   +67.208, E3 +66003.562}
SPL {X  -159.990, Y  +550.186, Z    +0.000, E1   +73.637, E3 +66028.967}
SPL {X  -159.493, Y  +364.902, Z    +0.000, E1   +74.541, E3 +66115.961}
SPL {X  -156.915, Y  +346.281, Z    +0.000, E1   +74.304, E3 +66129.557}
ENDSPLINE

SPLINE
SPL {X  -159.697, Y  +367.814, Z    +0.000, E1   +71.217, E3 +66146.875}
ENDSPLINE

SPLINE
SPL {X  -157.536, Y  +349.586, Z    +0.000, E1   +71.787, E3 +66154.173}
SPL {X  -154.855, Y  +337.291, Z    +0.000, E1   +72.155, E3 +66158.927}
SPL {X  -150.925, Y  +324.412, Z    +0.000, E1   +72.419, E3 +66164.821}
SPL {X  -146.819, Y  +313.931, Z    +0.000, E1   +72.621, E3 +66169.515}
SPL {X  -140.820, Y  +301.561, Z    +0.000, E1   +73.023, E3 +66173.431}
SPL {X  -136.475, Y  +294.006, Z    +0.000, E1   +72.670, E3 +66180.340}
SPL {X  -133.214, Y  +288.895, Z    +0.000, E1   +72.272, E3 +66185.988}
SPL {X  -129.829, Y  +284.006, Z    +0.000, E1   +71.844, E3 +66191.463}
SPL {X  -126.314, Y  +279.309, Z    +0.000, E1   +71.374, E3 +66196.755}
SPL {X  -122.705, Y  +274.834, Z    +0.000, E1   +70.869, E3 +66201.766}
SPL {X  -119.804, Y  +271.463, Z    +0.000, E1   +70.429, E3 +66205.485}
SPL {X   -77.409, Y  +237.483, Z    +0.000, E1   +59.013, E3 +66299.160}
ENDSPLINE

SPLINE
SPL {X  -103.775, Y  +255.731, Z    +0.000, E1   +56.205, E3 +66495.874}
SPL {X  -141.196, Y  +302.265, Z    +0.000, E1   +49.914, E3 +66533.359}
SPL {X  -155.405, Y  +339.473, Z    +0.000, E1   +34.418, E3 +66543.059}
SPL {X  -159.172, Y  +361.346, Z    +0.000, E1   +18.323, E3 +66545.484}
SPL {X  -159.962, Y  +374.520, Z    +0.000, E1    +5.534, E3 +66546.097}
SPL {X  -159.990, Y  +379.490, Z    +0.000, E1    +0.023, E3 +66546.154}
SPL {X  -159.990, Y  +381.667, Z    +0.000, E1    -4.707, E3 +66546.176}
SPL {X  -159.990, Y  +387.434, Z    +0.000, E1   -19.600, E3 +66546.359}
SPL {X  -159.990, Y  +395.000, Z    +0.000, E1   -38.121, E3 +66546.867}
SPL {X  -159.990, Y  +406.380, Z    +0.000, E1   -55.108, E3 +66548.309}
SPL {X  -159.990, Y  +426.664, Z    +0.000, E1   -66.963, E3 +66552.499}
SPL {X  -159.990, Y  +494.829, Z    +0.000, E1   -73.764, E3 +66574.263}
SPL {X  -158.798, Y  +695.991, Z    +0.000, E1   -74.986, E3 +66664.196}
SPL {X  -156.512, Y  +709.677, Z    +0.000, E1   -74.772, E3 +66674.340}
SPL {X  -153.684, Y  +720.975, Z    +0.000, E1   -74.508, E3 +66683.627}
SPL {X  -149.353, Y  +733.863, Z    +0.000, E1   -74.100, E3 +66695.215}
SPL {X  -145.190, Y  +743.705, Z    +0.000, E1   -73.640, E3 +66704.896}
SPL {X  -141.940, Y  +750.322, Z    +0.000, E1   -73.290, E3 +66711.663}
SPL {X  -138.555, Y  +756.496, Z    +0.000, E1   -72.905, E3 +66718.228}
SPL {X  -135.025, Y  +762.319, Z    +0.000, E1   -72.483, E3 +66724.607}
SPL {X  -131.747, Y  +767.272, Z    +0.000, E1   -72.071, E3 +66730.132}
SPL {X  -127.432, Y  +773.236, Z    +0.000, E1   -71.530, E3 +66736.818}
SPL {X  -124.036, Y  +777.554, Z    +0.000, E1   -71.026, E3 +66741.716}
SPL {X  -120.782, Y  +781.422, Z    +0.000, E1   -70.584, E3 +66745.974}
SPL {X   -74.295, Y  +818.193, Z    +0.000, E1   -57.793, E3 +66856.305}
ENDSPLINE

SPLINE
SPL {X  -105.102, Y  +797.125, Z    +0.000, E1   -55.734, E3 +67035.671}
SPL {X  -126.361, Y  +774.631, Z    +0.000, E1   -54.192, E3 +67061.339}
SPL {X  -145.777, Y  +742.423, Z    +0.000, E1   -46.722, E3 +67076.680}
SPL {X  -154.920, Y  +716.458, Z    +0.000, E1   -35.175, E3 +67082.735}
SPL {X  -158.252, Y  +700.019, Z    +0.000, E1   -24.087, E3 +67084.987}
SPL {X  -159.434, Y  +689.826, Z    +0.000, E1   -15.506, E3 +67085.805}
SPL {X  -159.958, Y  +679.684, Z    +0.000, E1    -5.688, E3 +67086.228}
SPL {X  -159.990, Y  +674.512, Z    +0.000, E1    -0.026, E3 +67086.293}
SPL {X  -159.990, Y  +672.767, Z    +0.000, E1    +3.705, E3 +67086.306}
SPL {X  -159.990, Y  +669.310, Z    +0.000, E1   +12.444, E3 +67086.380}
SPL {X  -159.990, Y  +665.511, Z    +0.000, E1   +22.359, E3 +67086.539}
SPL {X  -159.990, Y  +660.776, Z    +0.000, E1   +34.018, E3 +67086.845}
SPL {X  -159.990, Y  +655.863, Z    +0.000, E1   +43.768, E3 +67087.303}
SPL {X  -159.990, Y  +646.280, Z    +0.000, E1   +56.156, E3 +67088.592}
SPL {X  -159.990, Y  +625.549, Z    +0.000, E1   +67.208, E3 +67093.114}
SPL {X  -159.990, Y  +550.186, Z    +0.000, E1   +73.637, E3 +67118.520}
SPL {X  -159.878, Y  +371.520, Z    +0.000, E1   +74.559, E3 +67201.282}
SPL {X  -159.109, Y  +360.737, Z    +0.000, E1   +74.490, E3 +67208.406}
SPL {X  -156.915, Y  +346.281, Z    +0.000, E1   +74.304, E3 +67219.109}
ENDSPLINE

SPLINE
SPL {X  -159.697, Y  +367.814, Z    +0.000, E1   +71.217, E3 +67236.427}
ENDSPLINE

SPLINE
SPL {X  -156.028, Y  +342.114, Z    +0.000, E1   +72.020, E3 +67246.581}
SPL {X  -150.925, Y  +324.412, Z    +0.000, E1   +72.419, E3 +67254.374}
SPL {X  -146.819, Y  +313.931, Z    +0.000, E1   +72.621, E3 +67259.067}
SPL {X  -140.820, Y  +301.561, Z    +0.000, E1   +73.023, E3 +67262.983}
SPL {X  -136.475, Y  +294.006, Z    +0.000, E1   +72.670, E3 +67269.892}
SPL {X  -133.214, Y  +288.895, Z    +0.000, E1   +72.272, E3 +67275.540}
SPL {X  -129.829, Y  +284.006, Z    +0.000, E1   +71.844, E3 +67281.015}
SPL {X  -125.428, Y  +278.179, Z    +0.000, E1   +71.273, E3 +67287.552}
SPL {X  -120.729, Y  +272.518, Z    +0.000, E1   +70.593, E3 +67293.862}
SPL {X   -77.409, Y  +237.483, Z    +0.000, E1   +59.013, E3 +67388.713}
ENDSPLINE

SPLINE
SPL {X  -103.775, Y  +255.731, Z    +0.000, E1   +56.205, E3 +67585.426}
SPL {X  -141.196, Y  +302.265, Z    +0.000, E1   +49.914, E3 +67622.911}
SPL {X  -155.405, Y  +339.473, Z    +0.000, E1   +34.418, E3 +67632.611}
SPL {X  -159.172, Y  +361.346, Z    +0.000, E1   +18.323, E3 +67635.036}
SPL {X  -159.962, Y  +374.520, Z    +0.000, E1    +5.534, E3 +67635.649}
SPL {X  -159.990, Y  +379.490, Z    +0.000, E1    +0.023, E3 +67635.706}
SPL {X  -159.990, Y  +381.667, Z    +0.000, E1    -4.707, E3 +67635.728}
SPL {X  -159.990, Y  +385.814, Z    +0.000, E1   -15.621, E3 +67635.832}
SPL {X  -159.990, Y  +390.948, Z    +0.000, E1   -28.850, E3 +67636.108}
SPL {X  -159.990, Y  +399.006, Z    +0.000, E1   -45.565, E3 +67636.820}
SPL {X  -159.990, Y  +410.008, Z    +0.000, E1   -58.546, E3 +67638.430}
SPL {X  -159.990, Y  +430.714, Z    +0.000, E1   -67.965, E3 +67643.236}
SPL {X  -159.990, Y  +500.758, Z    +0.000, E1   -73.927, E3 +67665.911}
SPL {X  -158.798, Y  +695.991, Z    +0.000, E1   -74.986, E3 +67753.748}
SPL {X  -156.512, Y  +709.677, Z    +0.000, E1   -74.772, E3 +67763.892}
SPL {X  -153.684, Y  +720.975, Z    +0.000, E1   -74.508, E3 +67773.179}
SPL {X  -150.879, Y  +729.719, Z    +0.000, E1   -74.224, E3 +67780.973}
SPL {X  -148.237, Y  +736.689, Z    +0.000, E1   -73.960, E3 +67787.527}
SPL {X  -145.190, Y  +743.705, Z    +0.000, E1   -73.640, E3 +67794.448}
SPL {X  -141.940, Y  +750.322, Z    +0.000, E1   -73.290, E3 +67801.215}
SPL {X  -138.555, Y  +756.496, Z    +0.000, E1   -72.905, E3 +67807.780}
SPL {X  -135.025, Y  +762.319, Z    +0.000, E1   -72.483, E3 +67814.159}
SPL {X  -131.747, Y  +767.272, Z    +0.000, E1   -72.071, E3 +67819.684}
SPL {X  -127.432, Y  +773.236, Z    +0.000, E1   -71.530, E3 +67826.370}
SPL {X  -124.036, Y  +777.554, Z    +0.000, E1   -71.026, E3 +67831.268}
SPL {X  -120.782, Y  +781.422, Z    +0.000, E1   -70.584, E3 +67835.526}
SPL {X   -74.295, Y  +818.193, Z    +0.000, E1   -57.793, E3 +67945.857}
ENDSPLINE

SPLINE
SPL {X  -105.102, Y  +797.125, Z    +0.000, E1   -55.734, E3 +68125.224}
SPL {X  -126.361, Y  +774.631, Z    +0.000, E1   -54.192, E3 +68150.891}
SPL {X  -145.777, Y  +742.423, Z    +0.000, E1   -46.722, E3 +68166.232}
SPL {X  -154.920, Y  +716.458, Z    +0.000, E1   -35.175, E3 +68172.287}
SPL {X  -158.252, Y  +700.019, Z    +0.000, E1   -24.087, E3 +68174.539}
SPL {X  -159.676, Y  +686.525, Z    +0.000, E1   -12.514, E3 +68175.529}
SPL {X  -159.990, Y  +674.678, Z    +0.000, E1    -0.382, E3 +68175.844}
SPL {X  -159.990, Y  +672.767, Z    +0.000, E1    +3.705, E3 +68175.858}
SPL {X  -159.990, Y  +669.310, Z    +0.000, E1   +12.444, E3 +68175.932}
SPL {X  -159.990, Y  +665.511, Z    +0.000, E1   +22.359, E3 +68176.091}
SPL {X  -159.990, Y  +658.432, Z    +0.000, E1   +38.720, E3 +68176.616}
SPL {X  -159.990, Y  +646.280, Z    +0.000, E1   +56.156, E3 +68178.144}
SPL {X  -159.990, Y  +625.549, Z    +0.000, E1   +67.208, E3 +68182.666}
SPL {X  -159.990, Y  +550.186, Z    +0.000, E1   +73.637, E3 +68208.072}
SPL {X  -159.493, Y  +364.902, Z    +0.000, E1   +74.541, E3 +68295.065}
SPL {X  -156.915, Y  +346.281, Z    +0.000, E1   +74.304, E3 +68308.661}
ENDSPLINE

SPLINE
SPL {X  -159.697, Y  +367.814, Z    +0.000, E1   +71.217, E3 +68325.980}
ENDSPLINE

SPLINE
SPL {X  -156.028, Y  +342.114, Z    +0.000, E1   +72.020, E3 +68336.133}
SPL {X  -150.925, Y  +324.412, Z    +0.000, E1   +72.419, E3 +68343.926}
SPL {X  -144.972, Y  +309.824, Z    +0.000, E1   +72.799, E3 +68349.528}
SPL {X  -139.605, Y  +299.351, Z    +0.000, E1   +73.035, E3 +68353.660}
SPL {X  -136.475, Y  +294.006, Z    +0.000, E1   +72.670, E3 +68359.444}
SPL {X  -133.214, Y  +288.895, Z    +0.000, E1   +72.272, E3 +68365.092}
SPL {X  -129.829, Y  +284.006, Z    +0.000, E1   +71.844, E3 +68370.567}
SPL {X  -126.314, Y  +279.309, Z    +0.000, E1   +71.374, E3 +68375.859}
SPL {X  -122.705, Y  +274.834, Z    +0.000, E1   +70.869, E3 +68380.871}
SPL {X  -119.804, Y  +271.463, Z    +0.000, E1   +70.429, E3 +68384.589}
SPL {X   -77.409, Y  +237.483, Z    +0.000, E1   +59.013, E3 +68478.265}
ENDSPLINE

SPLINE
SPL {X  -103.775, Y  +255.731, Z    +0.000, E1   +56.205, E3 +68674.978}
SPL {X  -133.021, Y  +288.605, Z    +0.000, E1   +53.007, E3 +68706.435}
SPL {X  -149.384, Y  +320.219, Z    +0.000, E1   +43.953, E3 +68718.158}
SPL {X  -157.534, Y  +349.577, Z    +0.000, E1   +27.748, E3 +68723.510}
SPL {X  -159.460, Y  +364.489, Z    +0.000, E1   +15.407, E3 +68724.806}
SPL {X  -159.962, Y  +374.520, Z    +0.000, E1    +5.534, E3 +68725.201}
SPL {X  -159.990, Y  +379.490, Z    +0.000, E1    +0.023, E3 +68725.259}
SPL {X  -159.990, Y  +381.667, Z    +0.000, E1    -4.707, E3 +68725.281}
SPL {X  -159.990, Y  +387.434, Z    +0.000, E1   -19.600, E3 +68725.463}
SPL {X  -159.990, Y  +392.971, Z    +0.000, E1   -33.903, E3 +68725.796}
SPL {X  -159.990, Y  +399.006, Z    +0.000, E1   -45.565, E3 +68726.372}
SPL {X  -159.990, Y  +410.008, Z    +0.000, E1   -58.546, E3 +68727.983}
SPL {X  -159.990, Y  +426.664, Z    +0.000, E1   -66.963, E3 +68731.604}
SPL {X  -159.990, Y  +494.829, Z    +0.000, E1   -73.764, E3 +68753.368}
SPL {X  -158.798, Y  +695.991, Z    +0.000, E1   -74.986, E3 +68843.301}
SPL {X  -156.512, Y  +709.677, Z    +0.000, E1   -74.772, E3 +68853.444}
SPL {X  -153.684, Y  +720.975, Z    +0.000, E1   -74.508, E3 +68862.732}
SPL {X  -149.353, Y  +733.863, Z    +0.000, E1   -74.100, E3 +68874.319}
SPL {X  -145.190, Y  +743.705, Z    +0.000, E1   -73.640, E3 +68884.000}
SPL {X  -141.940, Y  +750.322, Z    +0.000, E1   -73.290, E3 +68890.767}
SPL {X  -138.555, Y  +756.496, Z    +0.000, E1   -72.905, E3 +68897.332}
SPL {X  -135.025, Y  +762.319, Z    +0.000, E1   -72.483, E3 +68903.712}
SPL {X  -131.747, Y  +767.272, Z    +0.000, E1   -72.071, E3 +68909.237}
SPL {X  -128.648, Y  +771.613, Z    +0.000, E1   -71.666, E3 +68914.129}
SPL {X  -125.012, Y  +776.344, Z    +0.000, E1   -71.184, E3 +68919.441}
SPL {X  -121.578, Y  +780.498, Z    +0.000, E1   -70.681, E3 +68924.084}
SPL {X  -119.460, Y  +782.925, Z    +0.000, E1   -70.353, E3 +68926.748}
SPL {X   -74.295, Y  +818.193, Z    +0.000, E1   -57.793, E3 +69035.409}
ENDSPLINE

SPLINE
SPL {X  -120.240, Y  +782.043, Z    +0.000, E1   -55.019, E3 +69233.905}
SPL {X  -145.777, Y  +742.423, Z    +0.000, E1   -46.722, E3 +69255.784}
SPL {X  -154.920, Y  +716.458, Z    +0.000, E1   -35.175, E3 +69261.839}
SPL {X  -159.063, Y  +693.702, Z    +0.000, E1   -19.028, E3 +69264.621}
SPL {X  -159.958, Y  +679.684, Z    +0.000, E1    -5.688, E3 +69265.333}
SPL {X  -159.990, Y  +674.512, Z    +0.000, E1    -0.026, E3 +69265.397}
SPL {X  -159.990, Y  +672.767, Z    +0.000, E1    +3.705, E3 +69265.411}
SPL {X  -159.990, Y  +669.310, Z    +0.000, E1   +12.444, E3 +69265.484}
SPL {X  -159.990, Y  +665.511, Z    +0.000, E1   +22.359, E3 +69265.643}
SPL {X  -159.990, Y  +658.432, Z    +0.000, E1   +38.720, E3 +69266.168}
SPL {X  -159.990, Y  +646.280, Z    +0.000, E1   +56.156, E3 +69267.697}
SPL {X  -159.990, Y  +625.549, Z    +0.000, E1   +67.208, E3 +69272.218}
SPL {X  -159.990, Y  +550.186, Z    +0.000, E1   +73.637, E3 +69297.624}
SPL {X  -159.878, Y  +371.520, Z    +0.000, E1   +74.559, E3 +69380.386}
SPL {X  -159.109, Y  +360.737, Z    +0.000, E1   +74.490, E3 +69387.510}
SPL {X  -156.915, Y  +346.281, Z    +0.000, E1   +74.304, E3 +69398.213}
ENDSPLINE

SPLINE
SPL {X  -159.697, Y  +367.814, Z    +0.000, E1   +71.217, E3 +69415.532}
ENDSPLINE

SPLINE
SPL {X  -157.536, Y  +349.586, Z    +0.000, E1   +71.787, E3 +69422.830}
SPL {X  -154.855, Y  +337.291, Z    +0.000, E1   +72.155, E3 +69427.584}
SPL {X  -150.925, Y  +324.412, Z    +0.000, E1   +72.419, E3 +69433.478}
SPL {X  -146.819, Y  +313.931, Z    +0.000, E1   +72.621, E3 +69438.171}
SPL {X  -140.820, Y  +301.561, Z    +0.000, E1   +73.023, E3 +69442.088}
SPL {X  -136.475, Y  +294.006, Z    +0.000, E1   +72.670, E3 +69448.997}
SPL {X  -133.214, Y  +288.895, Z    +0.000, E1   +72.272, E3 +69454.644}
SPL {X  -129.829, Y  +284.006, Z    +0.000, E1   +71.844, E3 +69460.119}
SPL {X  -126.314, Y  +279.309, Z    +0.000, E1   +71.374, E3 +69465.412}
SPL {X  -122.705, Y  +274.834, Z    +0.000, E1   +70.869, E3 +69470.423}
SPL {X  -119.804, Y  +271.463, Z    +0.000, E1   +70.429, E3 +69474.142}
SPL {X   -77.409, Y  +237.483, Z    +0.000, E1   +59.013, E3 +69567.817}
ENDSPLINE

SPLINE
SPL {X  -103.775, Y  +255.731, Z    +0.000, E1   +56.205, E3 +69764.530}
SPL {X  -141.196, Y  +302.265, Z    +0.000, E1   +49.914, E3 +69802.015}
SPL {X  -153.296, Y  +331.706, Z    +0.000, E1   +38.681, E3 +69810.435}
SPL {X  -157.534, Y  +349.577, Z    +0.000, E1   +27.748, E3 +69813.062}
SPL {X  -159.460, Y  +364.489, Z    +0.000, E1   +15.407, E3 +69814.358}
SPL {X  -159.962, Y  +374.520, Z    +0.000, E1    +5.534, E3 +69814.753}
SPL {X  -159.990, Y  +379.490, Z    +0.000, E1    +0.023, E3 +69814.811}
SPL {X  -159.990, Y  +381.667, Z    +0.000, E1    -4.707, E3 +69814.833}
SPL {X  -159.990, Y  +385.814, Z    +0.000, E1   -15.621, E3 +69814.937}
SPL {X  -159.990, Y  +390.948, Z    +0.000, E1   -28.850, E3 +69815.213}
SPL {X  -159.990, Y  +399.006, Z    +0.000, E1   -45.565, E3 +69815.925}
SPL {X  -159.990, Y  +410.008, Z    +0.000, E1   -58.546, E3 +69817.535}
SPL {X  -159.990, Y  +430.714, Z    +0.000, E1   -67.965, E3 +69822.340}
SPL {X  -159.990, Y  +500.758, Z    +0.000, E1   -73.927, E3 +69845.016}
SPL {X  -158.798, Y  +695.991, Z    +0.000, E1   -74.986, E3 +69932.853}
SPL {X  -156.512, Y  +709.677, Z    +0.000, E1   -74.772, E3 +69942.996}
SPL {X  -153.684, Y  +720.975, Z    +0.000, E1   -74.508, E3 +69952.284}
SPL {X  -150.879, Y  +729.719, Z    +0.000, E1   -74.224, E3 +69960.078}
SPL {X  -148.237, Y  +736.689, Z    +0.000, E1   -73.960, E3 +69966.632}
SPL {X  -145.190, Y  +743.705, Z    +0.000, E1   -73.640, E3 +69973.553}
SPL {X  -141.940, Y  +750.322, Z    +0.000, E1   -73.290, E3 +69980.319}
SPL {X  -138.555, Y  +756.496, Z    +0.000, E1   -72.905, E3 +69986.884}
SPL {X  -135.025, Y  +762.319, Z    +0.000, E1   -72.483, E3 +69993.264}
SPL {X  -131.747, Y  +767.272, Z    +0.000, E1   -72.071, E3 +69998.789}
SPL {X  -127.432, Y  +773.236, Z    +0.000, E1   -71.530, E3 +70005.474}
SPL {X  -124.036, Y  +777.554, Z    +0.000, E1   -71.026, E3 +70010.373}
SPL {X  -120.782, Y  +781.422, Z    +0.000, E1   -70.584, E3 +70014.631}
SPL {X   -74.295, Y  +818.193, Z    +0.000, E1   -57.793, E3 +70124.961}
ENDSPLINE

SPLINE
SPL {X  -120.240, Y  +782.043, Z    +0.000, E1   -55.019, E3 +70323.457}
SPL {X  -145.777, Y  +742.423, Z    +0.000, E1   -46.722, E3 +70345.337}
SPL {X  -154.920, Y  +716.458, Z    +0.000, E1   -35.175, E3 +70351.391}
SPL {X  -158.252, Y  +700.019, Z    +0.000, E1   -24.087, E3 +70353.643}
SPL {X  -159.676, Y  +686.525, Z    +0.000, E1   -12.514, E3 +70354.633}
SPL {X  -159.990, Y  +674.678, Z    +0.000, E1    -0.382, E3 +70354.948}
SPL {X  -159.990, Y  +672.767, Z    +0.000, E1    +3.705, E3 +70354.963}
SPL {X  -159.990, Y  +669.310, Z    +0.000, E1   +12.444, E3 +70355.037}
SPL {X  -159.990, Y  +665.511, Z    +0.000, E1   +22.359, E3 +70355.195}
SPL {X  -159.990, Y  +660.776, Z    +0.000, E1   +34.018, E3 +70355.502}
SPL {X  -159.990, Y  +655.863, Z    +0.000, E1   +43.768, E3 +70355.959}
SPL {X  -159.990, Y  +646.280, Z    +0.000, E1   +56.156, E3 +70357.249}
SPL {X  -159.990, Y  +625.549, Z    +0.000, E1   +67.208, E3 +70361.770}
SPL {X  -159.990, Y  +550.186, Z    +0.000, E1   +73.637, E3 +70387.176}
SPL {X  -159.878, Y  +371.520, Z    +0.000, E1   +74.559, E3 +70469.938}
SPL {X  -159.109, Y  +360.737, Z    +0.000, E1   +74.490, E3 +70477.063}
SPL {X  -156.915, Y  +346.281, Z    +0.000, E1   +74.304, E3 +70487.766}
ENDSPLINE

SPLINE
SPL {X  -159.697, Y  +367.814, Z    +0.000, E1   +71.217, E3 +70505.084}
ENDSPLINE

SPLINE
SPL {X  -157.536, Y  +349.586, Z    +0.000, E1   +71.787, E3 +70512.382}
SPL {X  -154.855, Y  +337.291, Z    +0.000, E1   +72.155, E3 +70517.136}
SPL {X  -150.925, Y  +324.412, Z    +0.000, E1   +72.419, E3 +70523.030}
SPL {X  -144.972, Y  +309.824, Z    +0.000, E1   +72.799, E3 +70528.632}
SPL {X  -139.605, Y  +299.351, Z    +0.000, E1   +73.035, E3 +70532.764}
SPL {X  -136.475, Y  +294.006, Z    +0.000, E1   +72.670, E3 +70538.549}
SPL {X  -133.214, Y  +288.895, Z    +0.000, E1   +72.272, E3 +70544.197}
SPL {X  -129.829, Y  +284.006, Z    +0.000, E1   +71.844, E3 +70549.672}
SPL {X  -126.314, Y  +279.309, Z    +0.000, E1   +71.374, E3 +70554.964}
SPL {X  -122.705, Y  +274.834, Z    +0.000, E1   +70.869, E3 +70559.975}
SPL {X  -119.804, Y  +271.463, Z    +0.000, E1   +70.429, E3 +70563.694}
SPL {X   -77.409, Y  +237.483, Z    +0.000, E1   +59.013, E3 +70657.369}
ENDSPLINE

SPLINE
SPL {X  -103.775, Y  +255.731, Z    +0.000, E1   +56.205, E3 +70854.083}
SPL {X  -141.196, Y  +302.265, Z    +0.000, E1   +49.914, E3 +70891.568}
SPL {X  -155.405, Y  +339.473, Z    +0.000, E1   +34.418, E3 +70901.268}
SPL {X  -158.399, Y  +354.990, Z    +0.000, E1   +23.559, E3 +70903.200}
SPL {X  -159.460, Y  +364.489, Z    +0.000, E1   +15.407, E3 +70903.910}
SPL {X  -159.962, Y  +374.520, Z    +0.000, E1    +5.534, E3 +70904.306}
SPL {X  -159.990, Y  +379.490, Z    +0.000, E1    +0.023, E3 +70904.363}
SPL {X  -159.990, Y  +381.667, Z    +0.000, E1    -4.707, E3 +70904.385}
SPL {X  -159.990, Y  +385.814, Z    +0.000, E1   -15.621, E3 +70904.489}
SPL {X  -159.990, Y  +390.948, Z    +0.000, E1   -28.850, E3 +70904.765}
SPL {X  -159.990, Y  +399.006, Z    +0.000, E1   -45.565, E3 +70905.477}
SPL {X  -159.990, Y  +410.008, Z    +0.000, E1   -58.546, E3 +70907.087}
SPL {X  -159.990, Y  +426.664, Z    +0.000, E1   -66.963, E3 +70910.708}
SPL {X  -159.990, Y  +494.829, Z    +0.000, E1   -73.764, E3 +70932.472}
SPL {X  -158.798, Y  +695.991, Z    +0.000, E1   -74.986, E3 +71022.405}
SPL {X  -156.512, Y  +709.677, Z    +0.000, E1   -74.772, E3 +71032.549}
SPL {X  -153.684, Y  +720.975, Z    +0.000, E1   -74.508, E3 +71041.836}
SPL {X  -149.353, Y  +733.863, Z    +0.000, E1   -74.100, E3 +71053.424}
SPL {X  -145.190, Y  +743.705, Z    +0.000, E1   -73.640, E3 +71063.105}
SPL {X  -141.940, Y  +750.322, Z    +0.000, E1   -73.290, E3 +71069.872}
SPL {X  -138.555, Y  +756.496, Z    +0.000, E1   -72.905, E3 +71076.437}
SPL {X  -135.025, Y  +762.319, Z    +0.000, E1   -72.483, E3 +71082.816}
SPL {X  -131.747, Y  +767.272, Z    +0.000, E1   -72.071, E3 +71088.341}
SPL {X  -128.648, Y  +771.613, Z    +0.000, E1   -71.666, E3 +71093.234}
SPL {X  -125.012, Y  +776.344, Z    +0.000, E1   -71.184, E3 +71098.545}
SPL {X  -120.782, Y  +781.422, Z    +0.000, E1   -70.584, E3 +71104.183}
SPL {X   -74.295, Y  +818.193, Z    +0.000, E1   -57.793, E3 +71214.514}
ENDSPLINE

SPLINE
SPL {X  -120.240, Y  +782.043, Z    +0.000, E1   -55.019, E3 +71413.009}
SPL {X  -145.777, Y  +742.423, Z    +0.000, E1   -46.722, E3 +71434.889}
SPL {X  -154.920, Y  +716.458, Z    +0.000, E1   -35.175, E3 +71440.944}
SPL {X  -159.063, Y  +693.702, Z    +0.000, E1   -19.028, E3 +71443.725}
SPL {X  -159.958, Y  +679.684, Z    +0.000, E1    -5.688, E3 +71444.437}
SPL {X  -159.990, Y  +674.512, Z    +0.000, E1    -0.026, E3 +71444.502}
SPL {X  -159.990, Y  +672.767, Z    +0.000, E1    +3.705, E3 +71444.515}
SPL {X  -159.990, Y  +669.310, Z    +0.000, E1   +12.444, E3 +71444.589}
SPL {X  -159.990, Y  +665.511, Z    +0.000, E1   +22.359, E3 +71444.748}
SPL {X  -159.990, Y  +658.432, Z    +0.000, E1   +38.720, E3 +71445.273}
SPL {X  -159.990, Y  +646.280, Z    +0.000, E1   +56.156, E3 +71446.801}
SPL {X  -159.990, Y  +625.549, Z    +0.000, E1   +67.208, E3 +71451.323}
SPL {X  -159.990, Y  +550.186, Z    +0.000, E1   +73.637, E3 +71476.728}
SPL {X  -159.493, Y  +364.902, Z    +0.000, E1   +74.541, E3 +71563.722}
SPL {X  -156.915, Y  +346.281, Z    +0.000, E1   +74.304, E3 +71577.318}
ENDSPLINE

SPLINE
SPL {X  -159.697, Y  +367.814, Z    +0.000, E1   +71.217, E3 +71594.636}
ENDSPLINE

SPLINE
SPL {X  -157.536, Y  +349.586, Z    +0.000, E1   +71.787, E3 +71601.934}
SPL {X  -154.855, Y  +337.291, Z    +0.000, E1   +72.155, E3 +71606.688}
SPL {X  -150.925, Y  +324.412, Z    +0.000, E1   +72.419, E3 +71612.583}
SPL {X  -146.819, Y  +313.931, Z    +0.000, E1   +72.621, E3 +71617.276}
SPL {X  -140.820, Y  +301.561, Z    +0.000, E1   +73.023, E3 +71621.192}
SPL {X  -136.475, Y  +294.006, Z    +0.000, E1   +72.670, E3 +71628.101}
SPL {X  -133.214, Y  +288.895, Z    +0.000, E1   +72.272, E3 +71633.749}
SPL {X  -129.829, Y  +284.006, Z    +0.000, E1   +71.844, E3 +71639.224}
SPL {X  -126.314, Y  +279.309, Z    +0.000, E1   +71.374, E3 +71644.516}
SPL {X  -122.705, Y  +274.834, Z    +0.000, E1   +70.869, E3 +71649.527}
SPL {X  -119.804, Y  +271.463, Z    +0.000, E1   +70.429, E3 +71653.246}
SPL {X   -77.409, Y  +237.483, Z    +0.000, E1   +59.013, E3 +71746.922}
ENDSPLINE

SPLINE
SPL {X  -103.775, Y  +255.731, Z    +0.000, E1   +56.205, E3 +71943.635}
SPL {X  -141.196, Y  +302.265, Z    +0.000, E1   +49.914, E3 +71981.120}
SPL {X  -155.405, Y  +339.473, Z    +0.000, E1   +34.418, E3 +71990.820}
SPL {X  -159.172, Y  +361.346, Z    +0.000, E1   +18.323, E3 +71993.245}
SPL {X  -159.962, Y  +374.520, Z    +0.000, E1    +5.534, E3 +71993.858}
SPL {X  -159.990, Y  +379.490, Z    +0.000, E1    +0.023, E3 +71993.915}
SPL {X  -159.990, Y  +381.667, Z    +0.000, E1    -4.707, E3 +71993.937}
SPL {X  -159.990, Y  +385.814, Z    +0.000, E1   -15.621, E3 +71994.041}
SPL {X  -159.990, Y  +390.948, Z    +0.000, E1   -28.850, E3 +71994.317}
SPL {X  -159.990, Y  +399.006, Z    +0.000, E1   -45.565, E3 +71995.029}
SPL {X  -159.990, Y  +410.008, Z    +0.000, E1   -58.546, E3 +71996.639}
SPL {X  -159.990, Y  +426.664, Z    +0.000, E1   -66.963, E3 +72000.261}
SPL {X  -159.990, Y  +494.829, Z    +0.000, E1   -73.764, E3 +72022.025}
SPL {X  -158.798, Y  +695.991, Z    +0.000, E1   -74.986, E3 +72111.957}
SPL {X  -156.512, Y  +709.677, Z    +0.000, E1   -74.772, E3 +72122.101}
SPL {X  -153.684, Y  +720.975, Z    +0.000, E1   -74.508, E3 +72131.388}
SPL {X  -149.353, Y  +733.863, Z    +0.000, E1   -74.100, E3 +72142.976}
SPL {X  -145.190, Y  +743.705, Z    +0.000, E1   -73.640, E3 +72152.657}
SPL {X  -141.940, Y  +750.322, Z    +0.000, E1   -73.290, E3 +72159.424}
SPL {X  -138.555, Y  +756.496, Z    +0.000, E1   -72.905, E3 +72165.989}
SPL {X  -135.025, Y  +762.319, Z    +0.000, E1   -72.483, E3 +72172.368}
SPL {X  -131.747, Y  +767.272, Z    +0.000, E1   -72.071, E3 +72177.893}
SPL {X  -128.648, Y  +771.613, Z    +0.000, E1   -71.666, E3 +72182.786}
SPL {X  -125.012, Y  +776.344, Z    +0.000, E1   -71.184, E3 +72188.097}
SPL {X  -120.782, Y  +781.422, Z    +0.000, E1   -70.584, E3 +72193.735}
SPL {X   -74.295, Y  +818.193, Z    +0.000, E1   -57.793, E3 +72304.066}
ENDSPLINE

SPLINE
SPL {X  -105.102, Y  +797.125, Z    +0.000, E1   -55.734, E3 +72483.432}
SPL {X  -126.361, Y  +774.631, Z    +0.000, E1   -54.192, E3 +72509.100}
SPL {X  -145.777, Y  +742.423, Z    +0.000, E1   -46.722, E3 +72524.441}
SPL {X  -154.920, Y  +716.458, Z    +0.000, E1   -35.175, E3 +72530.496}
SPL {X  -159.063, Y  +693.702, Z    +0.000, E1   -19.028, E3 +72533.277}
SPL {X  -159.958, Y  +679.684, Z    +0.000, E1    -5.688, E3 +72533.989}
SPL {X  -159.990, Y  +674.512, Z    +0.000, E1    -0.026, E3 +72534.054}
SPL {X  -159.990, Y  +672.767, Z    +0.000, E1    +3.705, E3 +72534.067}
SPL {X  -159.990, Y  +669.310, Z    +0.000, E1   +12.444, E3 +72534.141}
SPL {X  -159.990, Y  +665.511, Z    +0.000, E1   +22.359, E3 +72534.300}
SPL {X  -159.990, Y  +658.432, Z    +0.000, E1   +38.720, E3 +72534.825}
SPL {X  -159.990, Y  +646.280, Z    +0.000, E1   +56.156, E3 +72536.353}
SPL {X  -159.990, Y  +625.549, Z    +0.000, E1   +67.208, E3 +72540.875}
SPL {X  -159.990, Y  +550.186, Z    +0.000, E1   +73.637, E3 +72566.281}
SPL {X  -159.493, Y  +364.902, Z    +0.000, E1   +74.541, E3 +72653.274}
SPL {X  -156.915, Y  +346.281, Z    +0.000, E1   +74.304, E3 +72666.870}
ENDSPLINE

SPLINE
SPL {X  -159.697, Y  +367.814, Z    +0.000, E1   +71.217, E3 +72684.189}
ENDSPLINE

SPLINE
SPL {X  -156.028, Y  +342.114, Z    +0.000, E1   +72.020, E3 +72694.342}
SPL {X  -150.925, Y  +324.412, Z    +0.000, E1   +72.419, E3 +72702.135}
SPL {X  -144.972, Y  +309.824, Z    +0.000, E1   +72.799, E3 +72707.737}
ENDSPLINE

SLIN {X  -200.000, Y  +530.000, E1    +0.000}
HALT
END
